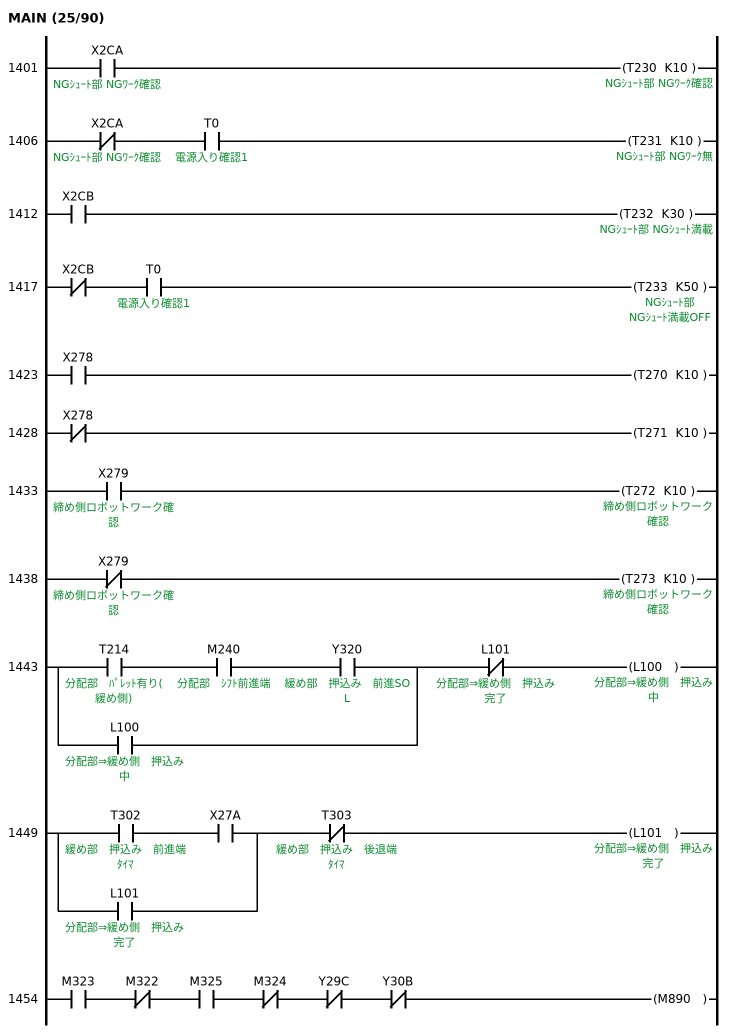
[picture p24: ladder of MAIN, rungs at steps 1401 to 1454]
1401  LD      X2CA  ; NGｼｭｰﾄ部 NGﾜｰｸ確認
      OUT     T230 K10  ; NGｼｭｰﾄ部 NGﾜｰｸ確認
1406  LDI     X2CA  ; NGｼｭｰﾄ部 NGﾜｰｸ確認
      AND     T0  ; 電源入り確認1
      OUT     T231 K10  ; NGｼｭｰﾄ部 NGﾜｰｸ無
1412  LD      X2CB
      OUT     T232 K30  ; NGｼｭｰﾄ部 NGｼｭｰﾄ満載
1417  LDI     X2CB
      AND     T0  ; 電源入り確認1
      OUT     T233 K50  ; NGｼｭｰﾄ部 NGｼｭｰﾄ満載OFF
1423  LD      X278
      OUT     T270 K10
1428  LDI     X278
      OUT     T271 K10
1433  LD      X279  ; 締め側ロボットワーク確認
      OUT     T272 K10  ; 締め側ロボットワーク確認
1438  LDI     X279  ; 締め側ロボットワーク確認
      OUT     T273 K10  ; 締め側ロボットワーク確認
1443  LD      T214  ; 分配部　ﾊﾟﾚｯﾄ有り(緩め側)
      AND     M240  ; 分配部　ｼﾌﾄ前進端
      AND     Y320  ; 緩め部　押込み　前進SOL
      OR      L100  ; 分配部⇒緩め側　押込み中
      ANI     L101  ; 分配部⇒緩め側　押込み完了
      OUT     L100  ; 分配部⇒緩め側　押込み中
1449  LD      T302  ; 緩め部　押込み　前進端　ﾀｲﾏ
      AND     X27A
      OR      L101  ; 分配部⇒緩め側　押込み完了
      ANI     T303  ; 緩め部　押込み　後退端　ﾀｲﾏ
      OUT     L101  ; 分配部⇒緩め側　押込み完了
1454  LD      M323
      ANI     M322
      AND     M325
      ANI     M324
      ANI     Y29C
      ANI     Y30B
      OUT     M890
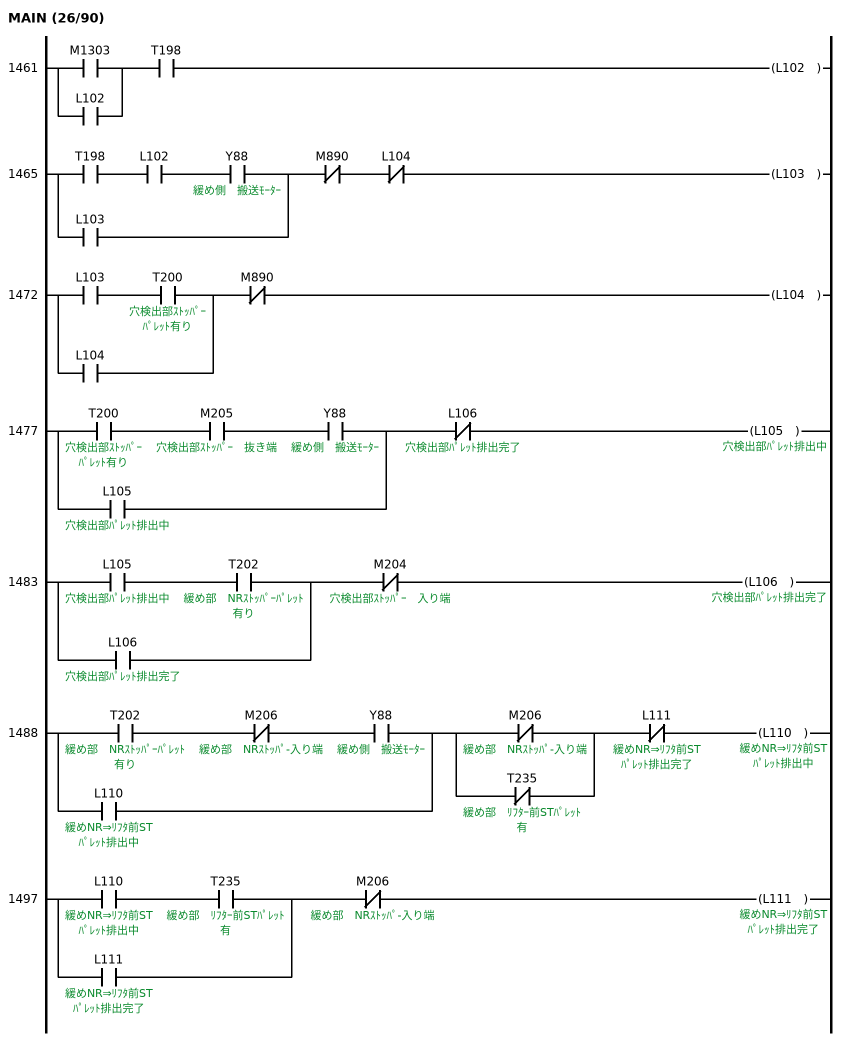
1461  LD      M1303
      OR      L102
      AND     T198
      OUT     L102
1465  LD      T198
      AND     L102
      AND     Y88  ; 緩め側　搬送ﾓｰﾀｰ
      OR      L103
      ANI     M890
      ANI     L104
      OUT     L103
1472  LD      L103
      AND     T200  ; 穴検出部ｽﾄｯﾊﾟｰ 　ﾊﾟﾚｯﾄ有り
      OR      L104
      ANI     M890
      OUT     L104
1477  LD      T200  ; 穴検出部ｽﾄｯﾊﾟｰ 　ﾊﾟﾚｯﾄ有り
      AND     M205  ; 穴検出部ｽﾄｯﾊﾟｰ　抜き端
      AND     Y88  ; 緩め側　搬送ﾓｰﾀｰ
      OR      L105  ; 穴検出部ﾊﾟﾚｯﾄ排出中
      ANI     L106  ; 穴検出部ﾊﾟﾚｯﾄ排出完了
      OUT     L105  ; 穴検出部ﾊﾟﾚｯﾄ排出中
1483  LD      L105  ; 穴検出部ﾊﾟﾚｯﾄ排出中
      AND     T202  ; 緩め部　NRｽﾄｯﾊﾟｰﾊﾟﾚｯﾄ有り
      OR      L106  ; 穴検出部ﾊﾟﾚｯﾄ排出完了
      ANI     M204  ; 穴検出部ｽﾄｯﾊﾟｰ　入り端
      OUT     L106  ; 穴検出部ﾊﾟﾚｯﾄ排出完了
1488  LD      T202  ; 緩め部　NRｽﾄｯﾊﾟｰﾊﾟﾚｯﾄ有り
      ANI     M206  ; 緩め部　NRｽﾄｯﾊﾟ-入り端
      AND     Y88  ; 緩め側　搬送ﾓｰﾀｰ
      OR      L110  ; 緩めNR⇒ﾘﾌﾀ前ST ﾊﾟﾚｯﾄ排出中
      LDI     M206  ; 緩め部　NRｽﾄｯﾊﾟ-入り端
      ORI     T235  ; 緩め部　ﾘﾌﾀｰ前STﾊﾟﾚｯﾄ有
      ANB
      ANI     L111  ; 緩めNR⇒ﾘﾌﾀ前ST ﾊﾟﾚｯﾄ排出完了
      OUT     L110  ; 緩めNR⇒ﾘﾌﾀ前ST ﾊﾟﾚｯﾄ排出中
1497  LD      L110  ; 緩めNR⇒ﾘﾌﾀ前ST ﾊﾟﾚｯﾄ排出中
      AND     T235  ; 緩め部　ﾘﾌﾀｰ前STﾊﾟﾚｯﾄ有
      OR      L111  ; 緩めNR⇒ﾘﾌﾀ前ST ﾊﾟﾚｯﾄ排出完了
      ANI     M206  ; 緩め部　NRｽﾄｯﾊﾟ-入り端
      OUT     L111  ; 緩めNR⇒ﾘﾌﾀ前ST ﾊﾟﾚｯﾄ排出完了
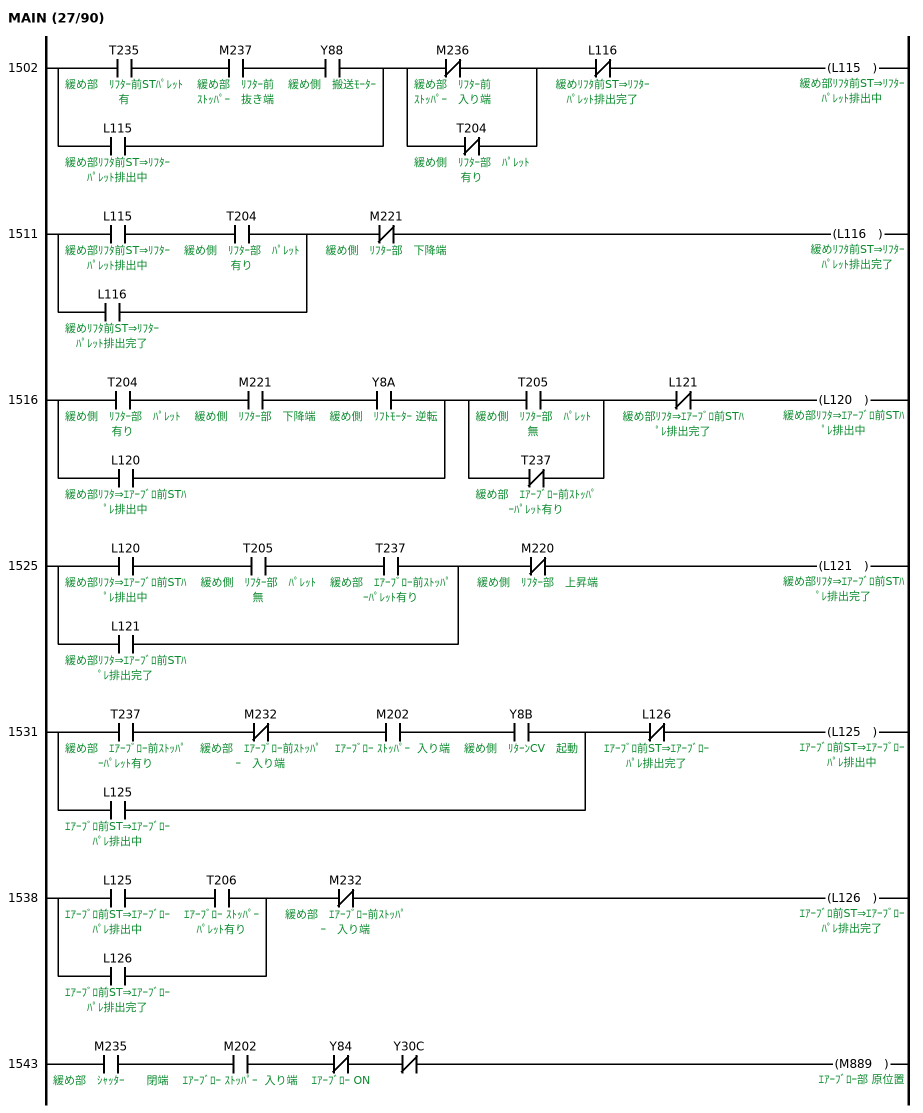
1502  LD      T235  ; 緩め部　ﾘﾌﾀｰ前STﾊﾟﾚｯﾄ有
      AND     M237  ; 緩め部　ﾘﾌﾀｰ前  ｽﾄｯﾊﾟｰ　抜き端
      AND     Y88  ; 緩め側　搬送ﾓｰﾀｰ
      OR      L115  ; 緩め部ﾘﾌﾀ前ST⇒ﾘﾌﾀｰ ﾊﾟﾚｯﾄ排出中
      LDI     M236  ; 緩め部　ﾘﾌﾀｰ前  ｽﾄｯﾊﾟｰ　入り端
      ORI     T204  ; 緩め側　ﾘﾌﾀｰ部　ﾊﾟﾚｯﾄ有り
      ANB
      ANI     L116  ; 緩めﾘﾌﾀ前ST⇒ﾘﾌﾀｰ ﾊﾟﾚｯﾄ排出完了
      OUT     L115  ; 緩め部ﾘﾌﾀ前ST⇒ﾘﾌﾀｰ ﾊﾟﾚｯﾄ排出中
1511  LD      L115  ; 緩め部ﾘﾌﾀ前ST⇒ﾘﾌﾀｰ ﾊﾟﾚｯﾄ排出中
      AND     T204  ; 緩め側　ﾘﾌﾀｰ部　ﾊﾟﾚｯﾄ有り
      OR      L116  ; 緩めﾘﾌﾀ前ST⇒ﾘﾌﾀｰ ﾊﾟﾚｯﾄ排出完了
      ANI     M221  ; 緩め側　ﾘﾌﾀｰ部　下降端
      OUT     L116  ; 緩めﾘﾌﾀ前ST⇒ﾘﾌﾀｰ ﾊﾟﾚｯﾄ排出完了
1516  LD      T204  ; 緩め側　ﾘﾌﾀｰ部　ﾊﾟﾚｯﾄ有り
      AND     M221  ; 緩め側　ﾘﾌﾀｰ部　下降端
      AND     Y8A  ; 緩め側　ﾘﾌﾄﾓｰﾀｰ 逆転
      OR      L120  ; 緩め部ﾘﾌﾀ⇒ｴｱｰﾌﾞﾛ前STﾊﾟﾚ排出中
      LD      T205  ; 緩め側　ﾘﾌﾀｰ部　ﾊﾟﾚｯﾄ無
      ORI     T237  ; 緩め部　ｴｱｰﾌﾞﾛｰ前ｽﾄｯﾊﾟｰﾊﾟﾚｯﾄ有り
      ANB
      ANI     L121  ; 緩め部ﾘﾌﾀ⇒ｴｱｰﾌﾞﾛ前STﾊﾟﾚ排出完了
      OUT     L120  ; 緩め部ﾘﾌﾀ⇒ｴｱｰﾌﾞﾛ前STﾊﾟﾚ排出中
1525  LD      L120  ; 緩め部ﾘﾌﾀ⇒ｴｱｰﾌﾞﾛ前STﾊﾟﾚ排出中
      AND     T205  ; 緩め側　ﾘﾌﾀｰ部　ﾊﾟﾚｯﾄ無
      AND     T237  ; 緩め部　ｴｱｰﾌﾞﾛｰ前ｽﾄｯﾊﾟｰﾊﾟﾚｯﾄ有り
      OR      L121  ; 緩め部ﾘﾌﾀ⇒ｴｱｰﾌﾞﾛ前STﾊﾟﾚ排出完了
      ANI     M220  ; 緩め側　ﾘﾌﾀｰ部　上昇端
      OUT     L121  ; 緩め部ﾘﾌﾀ⇒ｴｱｰﾌﾞﾛ前STﾊﾟﾚ排出完了
1531  LD      T237  ; 緩め部　ｴｱｰﾌﾞﾛｰ前ｽﾄｯﾊﾟｰﾊﾟﾚｯﾄ有り
      ANI     M232  ; 緩め部　ｴｱｰﾌﾞﾛｰ前ｽﾄｯﾊﾟｰ　入り端
      AND     M202  ; ｴｱｰﾌﾞﾛｰ ｽﾄｯﾊﾟｰ  入り端
      AND     Y8B  ; 緩め側　ﾘﾀｰﾝCV　起動
      OR      L125  ; ｴｱｰﾌﾞﾛ前ST⇒ｴｱｰﾌﾞﾛｰ ﾊﾟﾚ排出中
      ANI     L126  ; ｴｱｰﾌﾞﾛ前ST⇒ｴｱｰﾌﾞﾛｰ ﾊﾟﾚ排出完了
      OUT     L125  ; ｴｱｰﾌﾞﾛ前ST⇒ｴｱｰﾌﾞﾛｰ ﾊﾟﾚ排出中
1538  LD      L125  ; ｴｱｰﾌﾞﾛ前ST⇒ｴｱｰﾌﾞﾛｰ ﾊﾟﾚ排出中
      AND     T206  ; ｴｱｰﾌﾞﾛｰ ｽﾄｯﾊﾟｰ  ﾊﾟﾚｯﾄ有り
      OR      L126  ; ｴｱｰﾌﾞﾛ前ST⇒ｴｱｰﾌﾞﾛｰ ﾊﾟﾚ排出完了
      ANI     M232  ; 緩め部　ｴｱｰﾌﾞﾛｰ前ｽﾄｯﾊﾟｰ　入り端
      OUT     L126  ; ｴｱｰﾌﾞﾛ前ST⇒ｴｱｰﾌﾞﾛｰ ﾊﾟﾚ排出完了
1543  LD      M235  ; 緩め部　ｼｬｯﾀｰ　　閉端
      AND     M202  ; ｴｱｰﾌﾞﾛｰ ｽﾄｯﾊﾟｰ  入り端
      ANI     Y84  ; ｴｱｰﾌﾞﾛｰ ON
      ANI     Y30C
      OUT     M889  ; ｴｱｰﾌﾞﾛｰ部 原位置
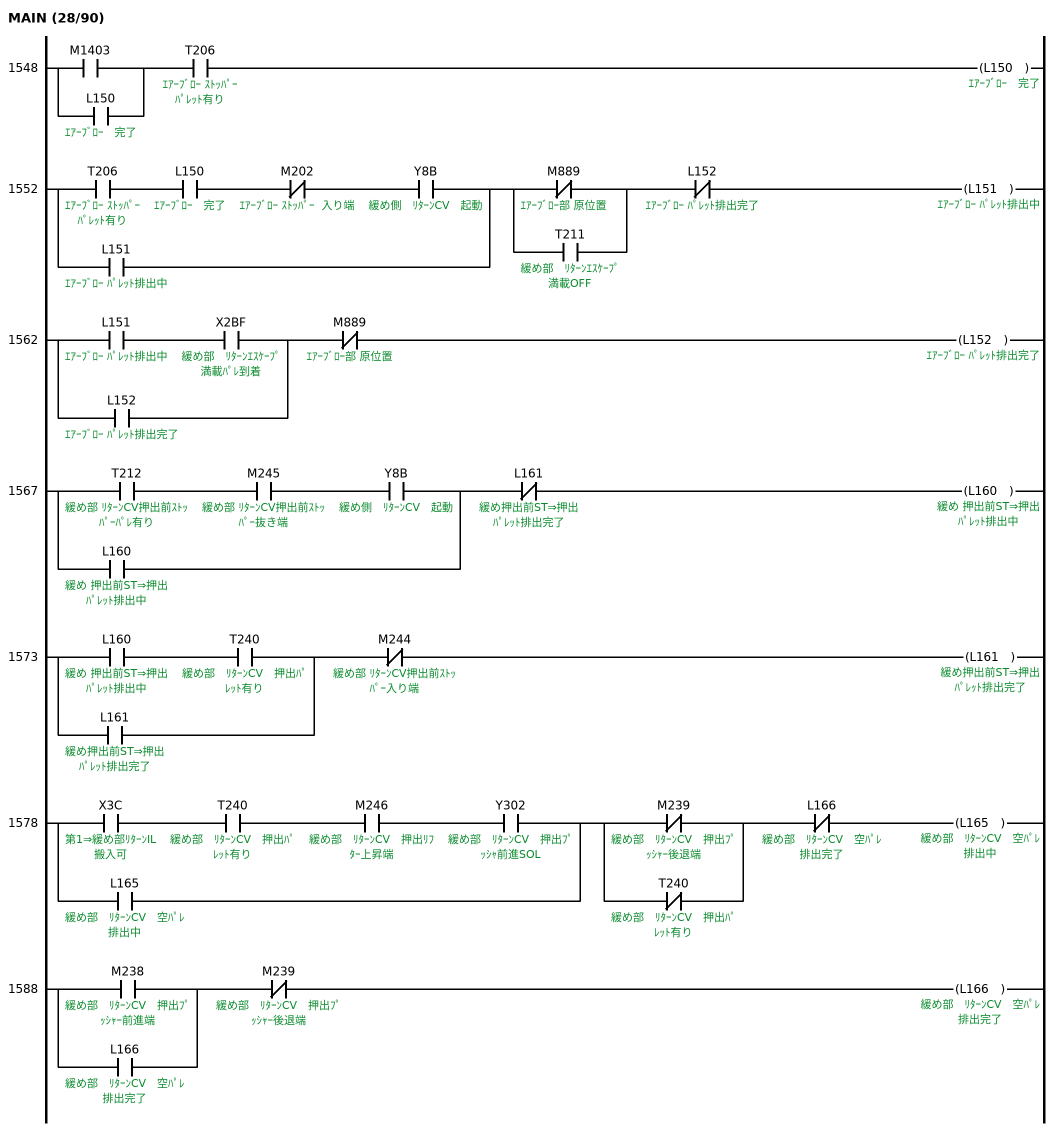
1548  LD      M1403
      OR      L150  ; ｴｱｰﾌﾞﾛｰ　完了
      AND     T206  ; ｴｱｰﾌﾞﾛｰ ｽﾄｯﾊﾟｰ  ﾊﾟﾚｯﾄ有り
      OUT     L150  ; ｴｱｰﾌﾞﾛｰ　完了
1552  LD      T206  ; ｴｱｰﾌﾞﾛｰ ｽﾄｯﾊﾟｰ  ﾊﾟﾚｯﾄ有り
      AND     L150  ; ｴｱｰﾌﾞﾛｰ　完了
      ANI     M202  ; ｴｱｰﾌﾞﾛｰ ｽﾄｯﾊﾟｰ  入り端
      AND     Y8B  ; 緩め側　ﾘﾀｰﾝCV　起動
      OR      L151  ; ｴｱｰﾌﾞﾛｰ ﾊﾟﾚｯﾄ排出中
      LDI     M889  ; ｴｱｰﾌﾞﾛｰ部 原位置
      OR      T211  ; 緩め部　ﾘﾀｰﾝｴｽｹｰﾌﾟ 満載OFF
      ANB
      ANI     L152  ; ｴｱｰﾌﾞﾛｰ ﾊﾟﾚｯﾄ排出完了
      OUT     L151  ; ｴｱｰﾌﾞﾛｰ ﾊﾟﾚｯﾄ排出中
1562  LD      L151  ; ｴｱｰﾌﾞﾛｰ ﾊﾟﾚｯﾄ排出中
      AND     X2BF  ; 緩め部　ﾘﾀｰﾝｴｽｹｰﾌﾟ 満載ﾊﾟﾚ到着
      OR      L152  ; ｴｱｰﾌﾞﾛｰ ﾊﾟﾚｯﾄ排出完了
      ANI     M889  ; ｴｱｰﾌﾞﾛｰ部 原位置
      OUT     L152  ; ｴｱｰﾌﾞﾛｰ ﾊﾟﾚｯﾄ排出完了
1567  LD      T212  ; 緩め部 ﾘﾀｰﾝCV押出前ｽﾄｯﾊﾟｰﾊﾟﾚ有り
      AND     M245  ; 緩め部 ﾘﾀｰﾝCV押出前ｽﾄｯﾊﾟｰ抜き端
      AND     Y8B  ; 緩め側　ﾘﾀｰﾝCV　起動
      OR      L160  ; 緩め 押出前ST⇒押出 ﾊﾟﾚｯﾄ排出中
      ANI     L161  ; 緩め押出前ST⇒押出 ﾊﾟﾚｯﾄ排出完了
      OUT     L160  ; 緩め 押出前ST⇒押出 ﾊﾟﾚｯﾄ排出中
1573  LD      L160  ; 緩め 押出前ST⇒押出 ﾊﾟﾚｯﾄ排出中
      AND     T240  ; 緩め部　ﾘﾀｰﾝCV　押出ﾊﾟﾚｯﾄ有り
      OR      L161  ; 緩め押出前ST⇒押出 ﾊﾟﾚｯﾄ排出完了
      ANI     M244  ; 緩め部 ﾘﾀｰﾝCV押出前ｽﾄｯﾊﾟｰ入り端
      OUT     L161  ; 緩め押出前ST⇒押出 ﾊﾟﾚｯﾄ排出完了
1578  LD      X3C  ; 第1⇒緩め部ﾘﾀｰﾝIL 搬入可
      AND     T240  ; 緩め部　ﾘﾀｰﾝCV　押出ﾊﾟﾚｯﾄ有り
      AND     M246  ; 緩め部　ﾘﾀｰﾝCV　押出ﾘﾌﾀｰ上昇端
      AND     Y302  ; 緩め部　ﾘﾀｰﾝCV　押出ﾌﾟｯｼｬ前進SOL
      OR      L165  ; 緩め部　ﾘﾀｰﾝCV　空ﾊﾟﾚ排出中
      LDI     M239  ; 緩め部　ﾘﾀｰﾝCV　押出ﾌﾟｯｼｬｰ後退端
      ORI     T240  ; 緩め部　ﾘﾀｰﾝCV　押出ﾊﾟﾚｯﾄ有り
      ANB
      ANI     L166  ; 緩め部　ﾘﾀｰﾝCV　空ﾊﾟﾚ排出完了
      OUT     L165  ; 緩め部　ﾘﾀｰﾝCV　空ﾊﾟﾚ排出中
1588  LD      M238  ; 緩め部　ﾘﾀｰﾝCV　押出ﾌﾟｯｼｬｰ前進端
      OR      L166  ; 緩め部　ﾘﾀｰﾝCV　空ﾊﾟﾚ排出完了
      ANI     M239  ; 緩め部　ﾘﾀｰﾝCV　押出ﾌﾟｯｼｬｰ後退端
      OUT     L166  ; 緩め部　ﾘﾀｰﾝCV　空ﾊﾟﾚ排出完了
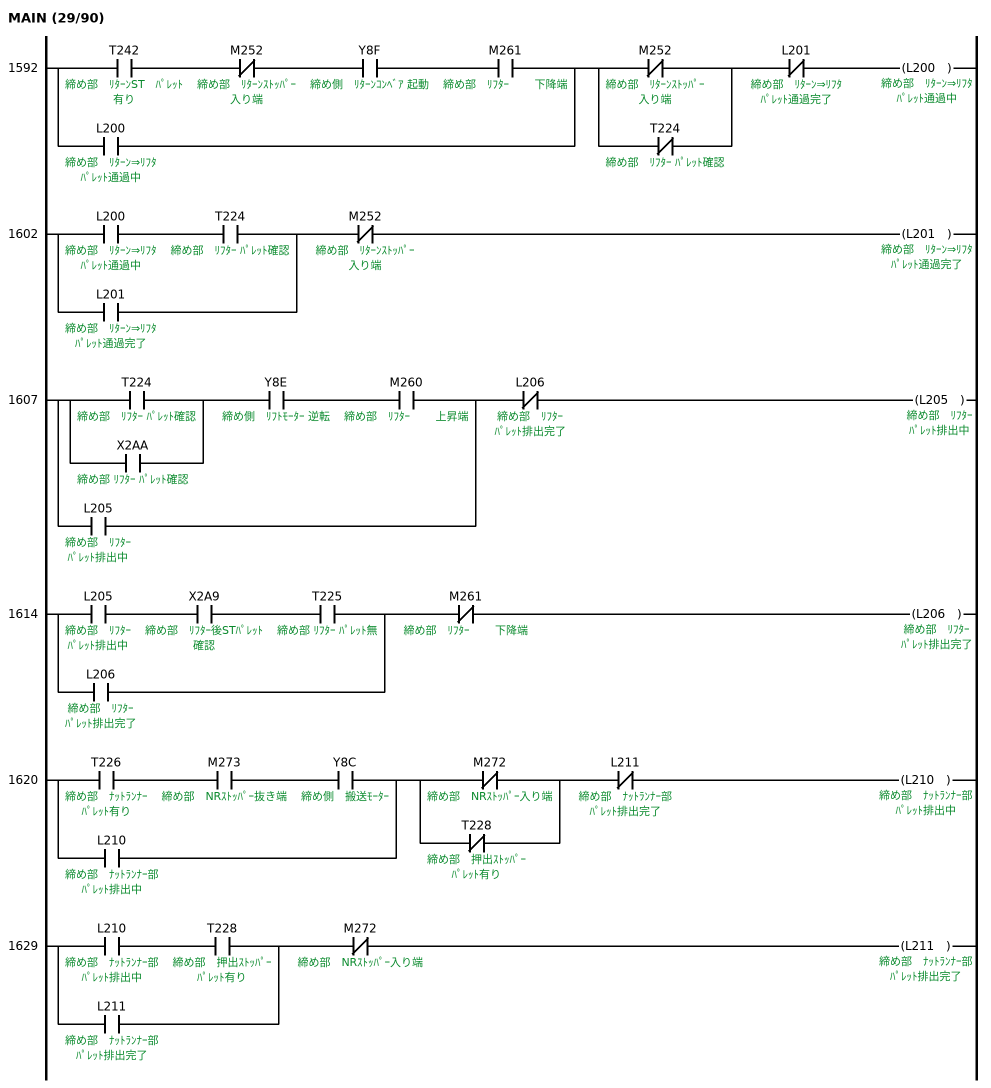
1592  LD      T242  ; 締め部　ﾘﾀｰﾝST　ﾊﾟﾚｯﾄ有り
      ANI     M252  ; 締め部　ﾘﾀｰﾝｽﾄｯﾊﾟｰ 入り端
      AND     Y8F  ; 締め側　ﾘﾀｰﾝｺﾝﾍﾞｱ 起動
      AND     M261  ; 締め部　ﾘﾌﾀｰ 　　下降端
      OR      L200  ; 締め部　ﾘﾀｰﾝ⇒ﾘﾌﾀ ﾊﾟﾚｯﾄ通過中
      LDI     M252  ; 締め部　ﾘﾀｰﾝｽﾄｯﾊﾟｰ 入り端
      ORI     T224  ; 締め部　ﾘﾌﾀｰ ﾊﾟﾚｯﾄ確認
      ANB
      ANI     L201  ; 締め部　ﾘﾀｰﾝ⇒ﾘﾌﾀ ﾊﾟﾚｯﾄ通過完了
      OUT     L200  ; 締め部　ﾘﾀｰﾝ⇒ﾘﾌﾀ ﾊﾟﾚｯﾄ通過中
1602  LD      L200  ; 締め部　ﾘﾀｰﾝ⇒ﾘﾌﾀ ﾊﾟﾚｯﾄ通過中
      AND     T224  ; 締め部　ﾘﾌﾀｰ ﾊﾟﾚｯﾄ確認
      OR      L201  ; 締め部　ﾘﾀｰﾝ⇒ﾘﾌﾀ ﾊﾟﾚｯﾄ通過完了
      ANI     M252  ; 締め部　ﾘﾀｰﾝｽﾄｯﾊﾟｰ 入り端
      OUT     L201  ; 締め部　ﾘﾀｰﾝ⇒ﾘﾌﾀ ﾊﾟﾚｯﾄ通過完了
1607  LD      T224  ; 締め部　ﾘﾌﾀｰ ﾊﾟﾚｯﾄ確認
      OR      X2AA  ; 締め部 ﾘﾌﾀｰ ﾊﾟﾚｯﾄ確認
      AND     Y8E  ; 締め側　ﾘﾌﾄﾓｰﾀｰ 逆転
      AND     M260  ; 締め部　ﾘﾌﾀｰ 　　上昇端
      OR      L205  ; 締め部　ﾘﾌﾀｰ ﾊﾟﾚｯﾄ排出中
      ANI     L206  ; 締め部　ﾘﾌﾀｰ ﾊﾟﾚｯﾄ排出完了
      OUT     L205  ; 締め部　ﾘﾌﾀｰ ﾊﾟﾚｯﾄ排出中
1614  LD      L205  ; 締め部　ﾘﾌﾀｰ ﾊﾟﾚｯﾄ排出中
      AND     X2A9  ; 締め部　ﾘﾌﾀｰ後STﾊﾟﾚｯﾄ確認
      AND     T225  ; 締め部 ﾘﾌﾀｰ ﾊﾟﾚｯﾄ無
      OR      L206  ; 締め部　ﾘﾌﾀｰ ﾊﾟﾚｯﾄ排出完了
      ANI     M261  ; 締め部　ﾘﾌﾀｰ 　　下降端
      OUT     L206  ; 締め部　ﾘﾌﾀｰ ﾊﾟﾚｯﾄ排出完了
1620  LD      T226  ; 締め部　ﾅｯﾄﾗﾝﾅｰ ﾊﾟﾚｯﾄ有り
      AND     M273  ; 締め部　NRｽﾄｯﾊﾟｰ抜き端
      AND     Y8C  ; 締め側　搬送ﾓｰﾀｰ
      OR      L210  ; 締め部　ﾅｯﾄﾗﾝﾅｰ部 ﾊﾟﾚｯﾄ排出中
      LDI     M272  ; 締め部　NRｽﾄｯﾊﾟｰ入り端
      ORI     T228  ; 締め部　押出ｽﾄｯﾊﾟｰ ﾊﾟﾚｯﾄ有り
      ANB
      ANI     L211  ; 締め部　ﾅｯﾄﾗﾝﾅｰ部 ﾊﾟﾚｯﾄ排出完了
      OUT     L210  ; 締め部　ﾅｯﾄﾗﾝﾅｰ部 ﾊﾟﾚｯﾄ排出中
1629  LD      L210  ; 締め部　ﾅｯﾄﾗﾝﾅｰ部 ﾊﾟﾚｯﾄ排出中
      AND     T228  ; 締め部　押出ｽﾄｯﾊﾟｰ ﾊﾟﾚｯﾄ有り
      OR      L211  ; 締め部　ﾅｯﾄﾗﾝﾅｰ部 ﾊﾟﾚｯﾄ排出完了
      ANI     M272  ; 締め部　NRｽﾄｯﾊﾟｰ入り端
      OUT     L211  ; 締め部　ﾅｯﾄﾗﾝﾅｰ部 ﾊﾟﾚｯﾄ排出完了
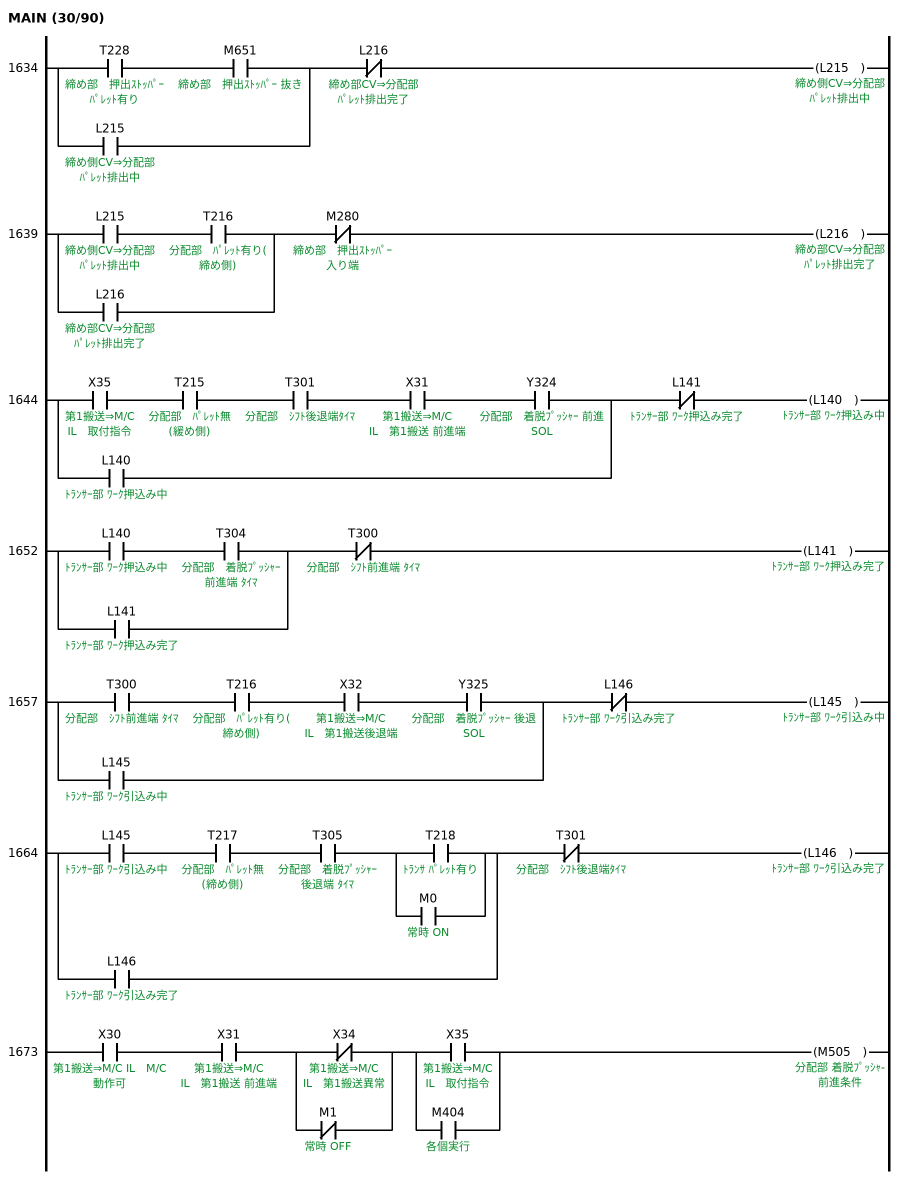
1634  LD      T228  ; 締め部　押出ｽﾄｯﾊﾟｰ ﾊﾟﾚｯﾄ有り
      AND     M651  ; 締め部　押出ｽﾄｯﾊﾟｰ 抜き
      OR      L215  ; 締め側CV⇒分配部 ﾊﾟﾚｯﾄ排出中
      ANI     L216  ; 締め部CV⇒分配部 ﾊﾟﾚｯﾄ排出完了
      OUT     L215  ; 締め側CV⇒分配部 ﾊﾟﾚｯﾄ排出中
1639  LD      L215  ; 締め側CV⇒分配部 ﾊﾟﾚｯﾄ排出中
      AND     T216  ; 分配部　ﾊﾟﾚｯﾄ有り(締め側)
      OR      L216  ; 締め部CV⇒分配部 ﾊﾟﾚｯﾄ排出完了
      ANI     M280  ; 締め部　押出ｽﾄｯﾊﾟｰ 入り端
      OUT     L216  ; 締め部CV⇒分配部 ﾊﾟﾚｯﾄ排出完了
1644  LD      X35  ; 第1搬送⇒M/C IL　取付指令
      AND     T215  ; 分配部　ﾊﾟﾚｯﾄ無 (緩め側)
      AND     T301  ; 分配部　ｼﾌﾄ後退端ﾀｲﾏ
      AND     X31  ; 第1搬送⇒M/C IL　第1搬送 前進端
      AND     Y324  ; 分配部　着脱ﾌﾟｯｼｬｰ 前進 SOL
      OR      L140  ; ﾄﾗﾝｻｰ部 ﾜｰｸ押込み中
      ANI     L141  ; ﾄﾗﾝｻｰ部 ﾜｰｸ押込み完了
      OUT     L140  ; ﾄﾗﾝｻｰ部 ﾜｰｸ押込み中
1652  LD      L140  ; ﾄﾗﾝｻｰ部 ﾜｰｸ押込み中
      AND     T304  ; 分配部　着脱ﾌﾟｯｼｬｰ 前進端 ﾀｲﾏ
      OR      L141  ; ﾄﾗﾝｻｰ部 ﾜｰｸ押込み完了
      ANI     T300  ; 分配部　ｼﾌﾄ前進端 ﾀｲﾏ
      OUT     L141  ; ﾄﾗﾝｻｰ部 ﾜｰｸ押込み完了
1657  LD      T300  ; 分配部　ｼﾌﾄ前進端 ﾀｲﾏ
      AND     T216  ; 分配部　ﾊﾟﾚｯﾄ有り(締め側)
      AND     X32  ; 第1搬送⇒M/C IL　第1搬送後退端
      AND     Y325  ; 分配部　着脱ﾌﾟｯｼｬｰ 後退 SOL
      OR      L145  ; ﾄﾗﾝｻｰ部 ﾜｰｸ引込み中
      ANI     L146  ; ﾄﾗﾝｻｰ部 ﾜｰｸ引込み完了
      OUT     L145  ; ﾄﾗﾝｻｰ部 ﾜｰｸ引込み中
1664  LD      L145  ; ﾄﾗﾝｻｰ部 ﾜｰｸ引込み中
      AND     T217  ; 分配部　ﾊﾟﾚｯﾄ無 (締め側)
      AND     T305  ; 分配部　着脱ﾌﾟｯｼｬｰ 後退端 ﾀｲﾏ
      LD      T218  ; ﾄﾗﾝｻ ﾊﾟﾚｯﾄ有り
      OR      M0  ; 常時 ON
      ANB
      OR      L146  ; ﾄﾗﾝｻｰ部 ﾜｰｸ引込み完了
      ANI     T301  ; 分配部　ｼﾌﾄ後退端ﾀｲﾏ
      OUT     L146  ; ﾄﾗﾝｻｰ部 ﾜｰｸ引込み完了
1673  LD      X30  ; 第1搬送⇒M/C IL　M/C 動作可
      AND     X31  ; 第1搬送⇒M/C IL　第1搬送 前進端
      LDI     X34  ; 第1搬送⇒M/C IL　第1搬送異常
      ORI     M1  ; 常時 OFF
      ANB
      LD      X35  ; 第1搬送⇒M/C IL　取付指令
      OR      M404  ; 各個実行
      ANB
      OUT     M505  ; 分配部 着脱ﾌﾟｯｼｬ- 前進条件
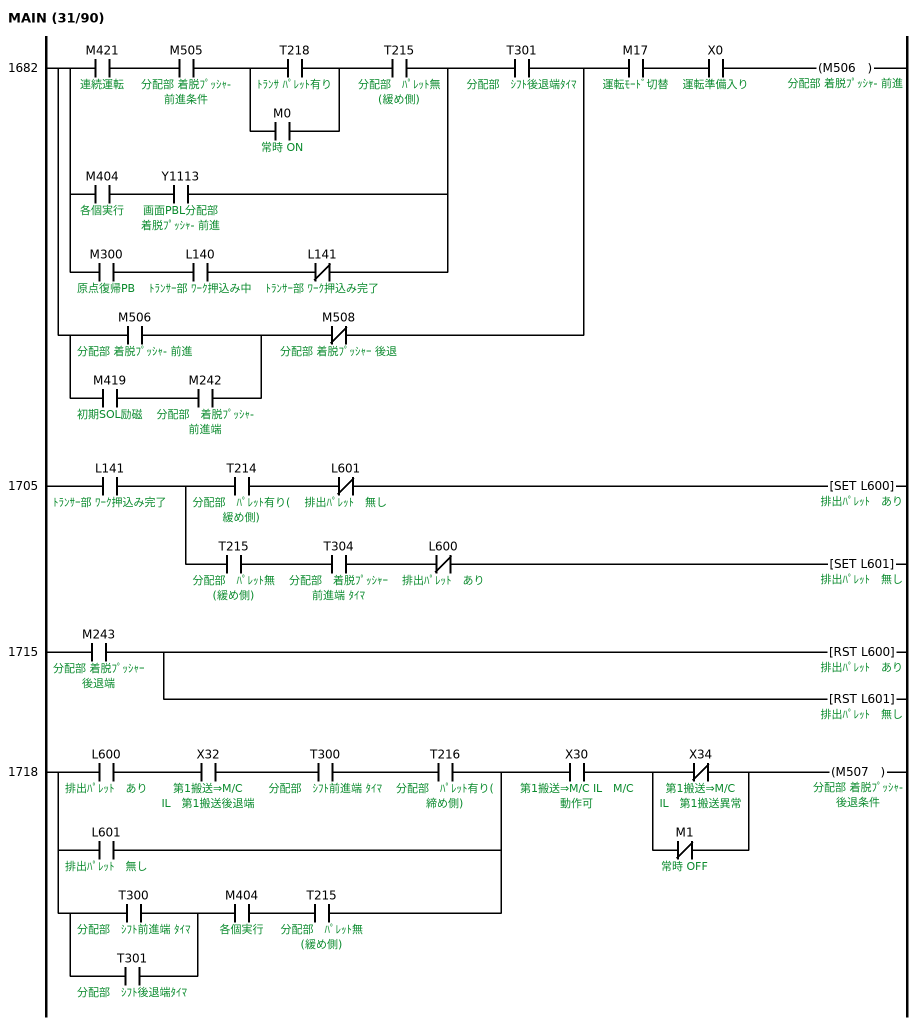
1682  LD      M421  ; 連続運転
      AND     M505  ; 分配部 着脱ﾌﾟｯｼｬ- 前進条件
      LD      T218  ; ﾄﾗﾝｻ ﾊﾟﾚｯﾄ有り
      OR      M0  ; 常時 ON
      ANB
      AND     T215  ; 分配部　ﾊﾟﾚｯﾄ無 (緩め側)
      LD      M404  ; 各個実行
      AND     Y1113  ; 画面PBL分配部 着脱ﾌﾟｯｼｬ- 前進
      ORB
      LD      M300  ; 原点復帰PB
      AND     L140  ; ﾄﾗﾝｻｰ部 ﾜｰｸ押込み中
      ANI     L141  ; ﾄﾗﾝｻｰ部 ﾜｰｸ押込み完了
      ORB
      AND     T301  ; 分配部　ｼﾌﾄ後退端ﾀｲﾏ
      LD      M506  ; 分配部 着脱ﾌﾟｯｼｬ- 前進
      LD      M419  ; 初期SOL励磁
      AND     M242  ; 分配部　着脱ﾌﾟｯｼｬ- 前進端
      ORB
      ANI     M508  ; 分配部 着脱ﾌﾟｯｼｬｰ 後退
      ORB
      AND     M17  ; 運転ﾓｰﾄﾞ切替
      AND     X0  ; 運転準備入り
      OUT     M506  ; 分配部 着脱ﾌﾟｯｼｬ- 前進
1705  LD      L141  ; ﾄﾗﾝｻｰ部 ﾜｰｸ押込み完了
      MPS
      AND     T214  ; 分配部　ﾊﾟﾚｯﾄ有り(緩め側)
      ANI     L601  ; 排出ﾊﾟﾚｯﾄ　無し
      SET     L600  ; 排出ﾊﾟﾚｯﾄ　あり
      MPP
      AND     T215  ; 分配部　ﾊﾟﾚｯﾄ無 (緩め側)
      AND     T304  ; 分配部　着脱ﾌﾟｯｼｬｰ 前進端 ﾀｲﾏ
      ANI     L600  ; 排出ﾊﾟﾚｯﾄ　あり
      SET     L601  ; 排出ﾊﾟﾚｯﾄ　無し
1715  LD      M243  ; 分配部 着脱ﾌﾟｯｼｬｰ 後退端
      RST     L600  ; 排出ﾊﾟﾚｯﾄ　あり
      RST     L601  ; 排出ﾊﾟﾚｯﾄ　無し
1718  LD      L600  ; 排出ﾊﾟﾚｯﾄ　あり
      AND     X32  ; 第1搬送⇒M/C IL　第1搬送後退端
      AND     T300  ; 分配部　ｼﾌﾄ前進端 ﾀｲﾏ
      AND     T216  ; 分配部　ﾊﾟﾚｯﾄ有り(締め側)
      OR      L601  ; 排出ﾊﾟﾚｯﾄ　無し
      LD      T300  ; 分配部　ｼﾌﾄ前進端 ﾀｲﾏ
      OR      T301  ; 分配部　ｼﾌﾄ後退端ﾀｲﾏ
      AND     M404  ; 各個実行
      AND     T215  ; 分配部　ﾊﾟﾚｯﾄ無 (緩め側)
      ORB
      AND     X30  ; 第1搬送⇒M/C IL　M/C 動作可
      LDI     X34  ; 第1搬送⇒M/C IL　第1搬送異常
      ORI     M1  ; 常時 OFF
      ANB
      OUT     M507  ; 分配部 着脱ﾌﾟｯｼｬ-後退条件
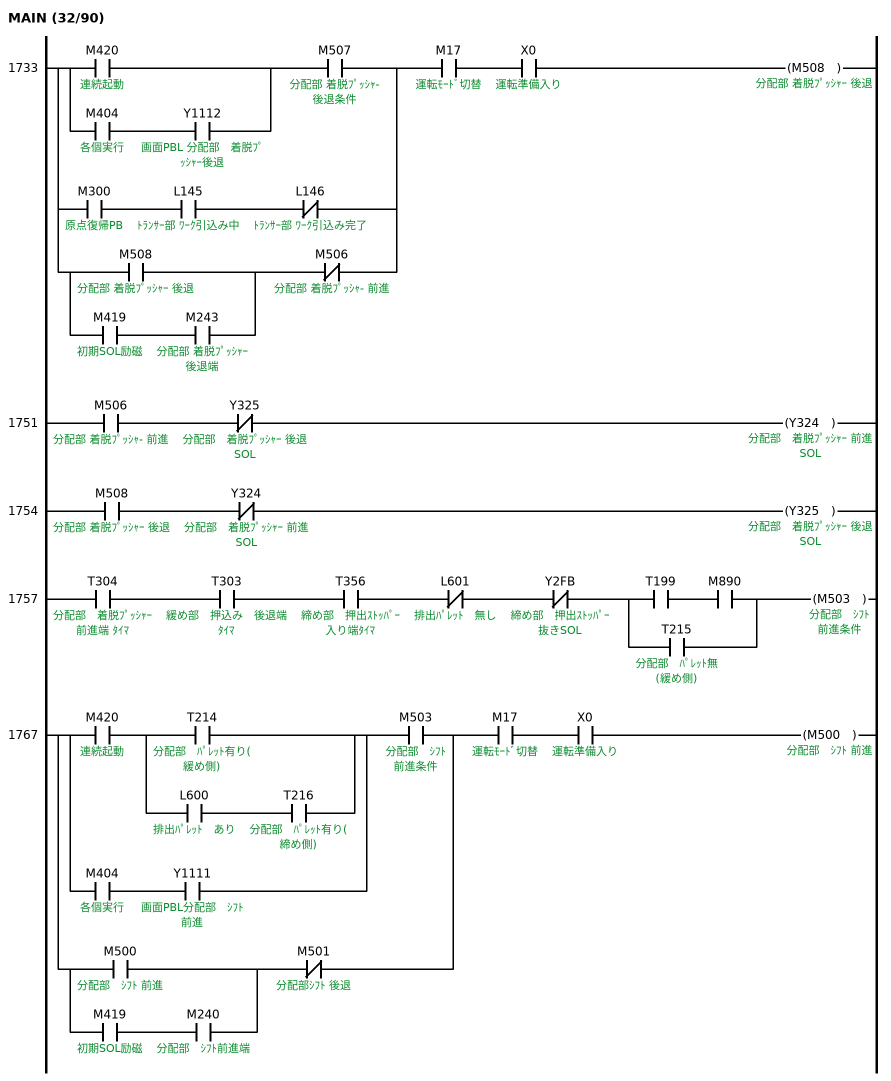
1733  LD      M420  ; 連続起動
      LD      M404  ; 各個実行
      AND     Y1112  ; 画面PBL 分配部　着脱ﾌﾟｯｼｬｰ後退
      ORB
      AND     M507  ; 分配部 着脱ﾌﾟｯｼｬ-後退条件
      LD      M300  ; 原点復帰PB
      AND     L145  ; ﾄﾗﾝｻｰ部 ﾜｰｸ引込み中
      ANI     L146  ; ﾄﾗﾝｻｰ部 ﾜｰｸ引込み完了
      ORB
      LD      M508  ; 分配部 着脱ﾌﾟｯｼｬｰ 後退
      LD      M419  ; 初期SOL励磁
      AND     M243  ; 分配部 着脱ﾌﾟｯｼｬｰ 後退端
      ORB
      ANI     M506  ; 分配部 着脱ﾌﾟｯｼｬ- 前進
      ORB
      AND     M17  ; 運転ﾓｰﾄﾞ切替
      AND     X0  ; 運転準備入り
      OUT     M508  ; 分配部 着脱ﾌﾟｯｼｬｰ 後退
1751  LD      M506  ; 分配部 着脱ﾌﾟｯｼｬ- 前進
      ANI     Y325  ; 分配部　着脱ﾌﾟｯｼｬｰ 後退 SOL
      OUT     Y324  ; 分配部　着脱ﾌﾟｯｼｬｰ 前進 SOL
1754  LD      M508  ; 分配部 着脱ﾌﾟｯｼｬｰ 後退
      ANI     Y324  ; 分配部　着脱ﾌﾟｯｼｬｰ 前進 SOL
      OUT     Y325  ; 分配部　着脱ﾌﾟｯｼｬｰ 後退 SOL
1757  LD      T304  ; 分配部　着脱ﾌﾟｯｼｬｰ 前進端 ﾀｲﾏ
      AND     T303  ; 緩め部　押込み　後退端　ﾀｲﾏ
      AND     T356  ; 締め部　押出ｽﾄｯﾊﾟｰ 入り端ﾀｲﾏ
      ANI     L601  ; 排出ﾊﾟﾚｯﾄ　無し
      ANI     Y2FB  ; 締め部　押出ｽﾄｯﾊﾟｰ 抜きSOL
      LD      T199
      AND     M890
      OR      T215  ; 分配部　ﾊﾟﾚｯﾄ無 (緩め側)
      ANB
      OUT     M503  ; 分配部　ｼﾌﾄ 　　前進条件
1767  LD      M420  ; 連続起動
      LD      T214  ; 分配部　ﾊﾟﾚｯﾄ有り(緩め側)
      LD      L600  ; 排出ﾊﾟﾚｯﾄ　あり
      AND     T216  ; 分配部　ﾊﾟﾚｯﾄ有り(締め側)
      ORB
      ANB
      LD      M404  ; 各個実行
      AND     Y1111  ; 画面PBL分配部　ｼﾌﾄ 前進
      ORB
      AND     M503  ; 分配部　ｼﾌﾄ 　　前進条件
      LD      M500  ; 分配部　ｼﾌﾄ 前進
      LD      M419  ; 初期SOL励磁
      AND     M240  ; 分配部　ｼﾌﾄ前進端
      ORB
      ANI     M501  ; 分配部ｼﾌﾄ 後退
      ORB
      AND     M17  ; 運転ﾓｰﾄﾞ切替
      AND     X0  ; 運転準備入り
      OUT     M500  ; 分配部　ｼﾌﾄ 前進
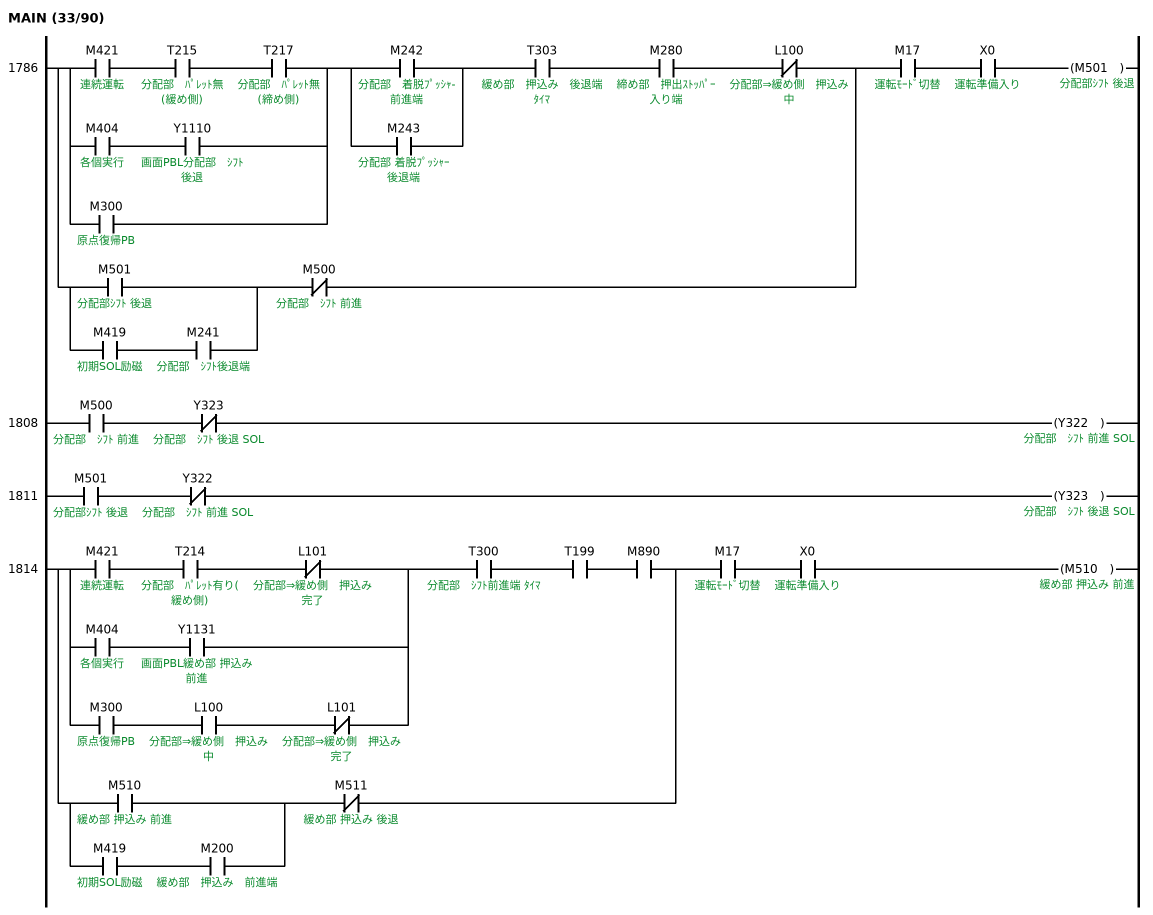
1786  LD      M421  ; 連続運転
      AND     T215  ; 分配部　ﾊﾟﾚｯﾄ無 (緩め側)
      AND     T217  ; 分配部　ﾊﾟﾚｯﾄ無 (締め側)
      LD      M404  ; 各個実行
      AND     Y1110  ; 画面PBL分配部　ｼﾌﾄ 後退
      ORB
      OR      M300  ; 原点復帰PB
      LD      M242  ; 分配部　着脱ﾌﾟｯｼｬ- 前進端
      OR      M243  ; 分配部 着脱ﾌﾟｯｼｬｰ 後退端
      ANB
      AND     T303  ; 緩め部　押込み　後退端　ﾀｲﾏ
      AND     M280  ; 締め部　押出ｽﾄｯﾊﾟｰ 入り端
      ANI     L100  ; 分配部⇒緩め側　押込み中
      LD      M501  ; 分配部ｼﾌﾄ 後退
      LD      M419  ; 初期SOL励磁
      AND     M241  ; 分配部　ｼﾌﾄ後退端
      ORB
      ANI     M500  ; 分配部　ｼﾌﾄ 前進
      ORB
      AND     M17  ; 運転ﾓｰﾄﾞ切替
      AND     X0  ; 運転準備入り
      OUT     M501  ; 分配部ｼﾌﾄ 後退
1808  LD      M500  ; 分配部　ｼﾌﾄ 前進
      ANI     Y323  ; 分配部　ｼﾌﾄ 後退 SOL
      OUT     Y322  ; 分配部　ｼﾌﾄ 前進 SOL
1811  LD      M501  ; 分配部ｼﾌﾄ 後退
      ANI     Y322  ; 分配部　ｼﾌﾄ 前進 SOL
      OUT     Y323  ; 分配部　ｼﾌﾄ 後退 SOL
1814  LD      M421  ; 連続運転
      AND     T214  ; 分配部　ﾊﾟﾚｯﾄ有り(緩め側)
      ANI     L101  ; 分配部⇒緩め側　押込み完了
      LD      M404  ; 各個実行
      AND     Y1131  ; 画面PBL緩め部 押込み 前進
      ORB
      LD      M300  ; 原点復帰PB
      AND     L100  ; 分配部⇒緩め側　押込み中
      ANI     L101  ; 分配部⇒緩め側　押込み完了
      ORB
      AND     T300  ; 分配部　ｼﾌﾄ前進端 ﾀｲﾏ
      AND     T199
      AND     M890
      LD      M510  ; 緩め部 押込み 前進
      LD      M419  ; 初期SOL励磁
      AND     M200  ; 緩め部　押込み　前進端
      ORB
      ANI     M511  ; 緩め部 押込み 後退
      ORB
      AND     M17  ; 運転ﾓｰﾄﾞ切替
      AND     X0  ; 運転準備入り
      OUT     M510  ; 緩め部 押込み 前進
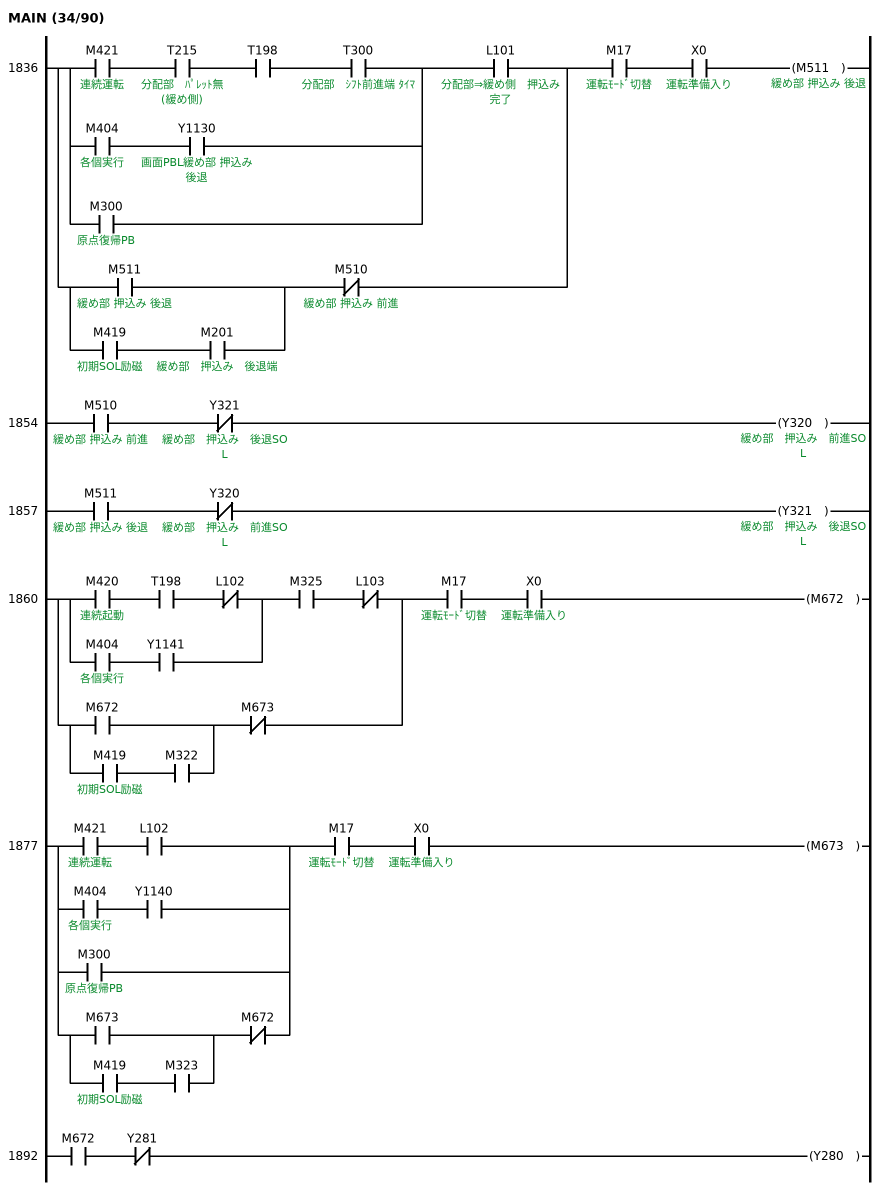
1836  LD      M421  ; 連続運転
      AND     T215  ; 分配部　ﾊﾟﾚｯﾄ無 (緩め側)
      AND     T198
      AND     T300  ; 分配部　ｼﾌﾄ前進端 ﾀｲﾏ
      LD      M404  ; 各個実行
      AND     Y1130  ; 画面PBL緩め部 押込み 後退
      ORB
      OR      M300  ; 原点復帰PB
      AND     L101  ; 分配部⇒緩め側　押込み完了
      LD      M511  ; 緩め部 押込み 後退
      LD      M419  ; 初期SOL励磁
      AND     M201  ; 緩め部　押込み　後退端
      ORB
      ANI     M510  ; 緩め部 押込み 前進
      ORB
      AND     M17  ; 運転ﾓｰﾄﾞ切替
      AND     X0  ; 運転準備入り
      OUT     M511  ; 緩め部 押込み 後退
1854  LD      M510  ; 緩め部 押込み 前進
      ANI     Y321  ; 緩め部　押込み　後退SOL
      OUT     Y320  ; 緩め部　押込み　前進SOL
1857  LD      M511  ; 緩め部 押込み 後退
      ANI     Y320  ; 緩め部　押込み　前進SOL
      OUT     Y321  ; 緩め部　押込み　後退SOL
1860  LD      M420  ; 連続起動
      AND     T198
      ANI     L102
      LD      M404  ; 各個実行
      AND     Y1141
      ORB
      AND     M325
      ANI     L103
      LD      M672
      LD      M419  ; 初期SOL励磁
      AND     M322
      ORB
      ANI     M673
      ORB
      AND     M17  ; 運転ﾓｰﾄﾞ切替
      AND     X0  ; 運転準備入り
      OUT     M672
1877  LD      M421  ; 連続運転
      AND     L102
      LD      M404  ; 各個実行
      AND     Y1140
      ORB
      OR      M300  ; 原点復帰PB
      LD      M673
      LD      M419  ; 初期SOL励磁
      AND     M323
      ORB
      ANI     M672
      ORB
      AND     M17  ; 運転ﾓｰﾄﾞ切替
      AND     X0  ; 運転準備入り
      OUT     M673
1892  LD      M672
      ANI     Y281
      OUT     Y280
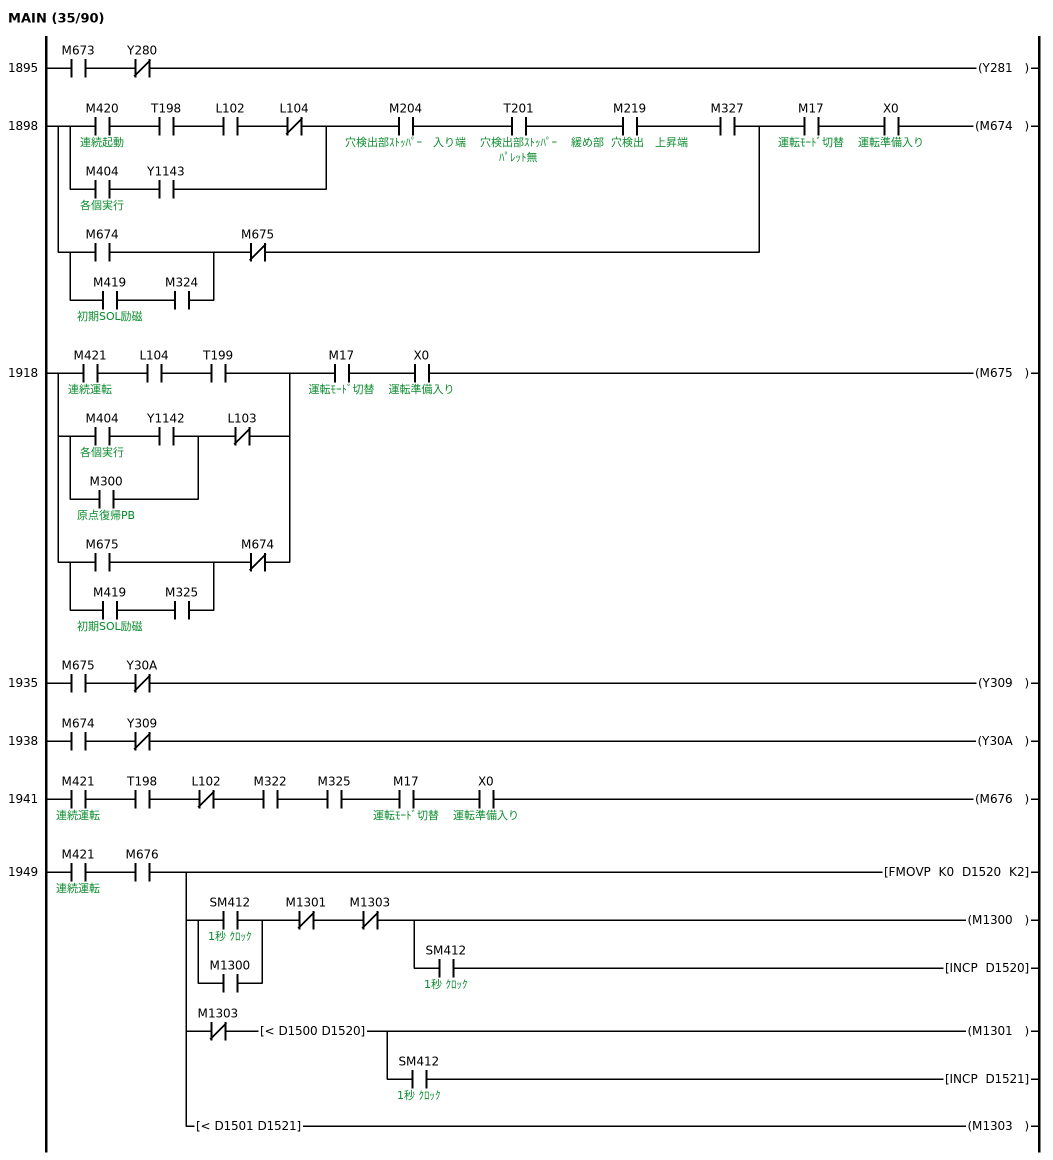
1895  LD      M673
      ANI     Y280
      OUT     Y281
1898  LD      M420  ; 連続起動
      AND     T198
      AND     L102
      ANI     L104
      LD      M404  ; 各個実行
      AND     Y1143
      ORB
      AND     M204  ; 穴検出部ｽﾄｯﾊﾟｰ　入り端
      AND     T201  ; 穴検出部ｽﾄｯﾊﾟｰ 　ﾊﾟﾚｯﾄ無
      AND     M219  ; 緩め部  穴検出　上昇端
      AND     M327
      LD      M674
      LD      M419  ; 初期SOL励磁
      AND     M324
      ORB
      ANI     M675
      ORB
      AND     M17  ; 運転ﾓｰﾄﾞ切替
      AND     X0  ; 運転準備入り
      OUT     M674
1918  LD      M421  ; 連続運転
      AND     L104
      AND     T199
      LD      M404  ; 各個実行
      AND     Y1142
      OR      M300  ; 原点復帰PB
      ANI     L103
      ORB
      LD      M675
      LD      M419  ; 初期SOL励磁
      AND     M325
      ORB
      ANI     M674
      ORB
      AND     M17  ; 運転ﾓｰﾄﾞ切替
      AND     X0  ; 運転準備入り
      OUT     M675
1935  LD      M675
      ANI     Y30A
      OUT     Y309
1938  LD      M674
      ANI     Y309
      OUT     Y30A
1941  LD      M421  ; 連続運転
      AND     T198
      ANI     L102
      AND     M322
      AND     M325
      AND     M17  ; 運転ﾓｰﾄﾞ切替
      AND     X0  ; 運転準備入り
      OUT     M676
1949  LD      M421  ; 連続運転
      AND     M676
      FMOVP   K0 D1520 K2
      MPS
      LD      SM412  ; 1秒 ｸﾛｯｸ
      OR      M1300
      ANB
      ANI     M1301
      ANI     M1303
      OUT     M1300
      AND     SM412  ; 1秒 ｸﾛｯｸ
      INCP    D1520
      MRD
      ANI     M1303
      AND<    D1500 D1520
      OUT     M1301
      AND     SM412  ; 1秒 ｸﾛｯｸ
      INCP    D1521
      MPP
      AND<    D1501 D1521
      OUT     M1303
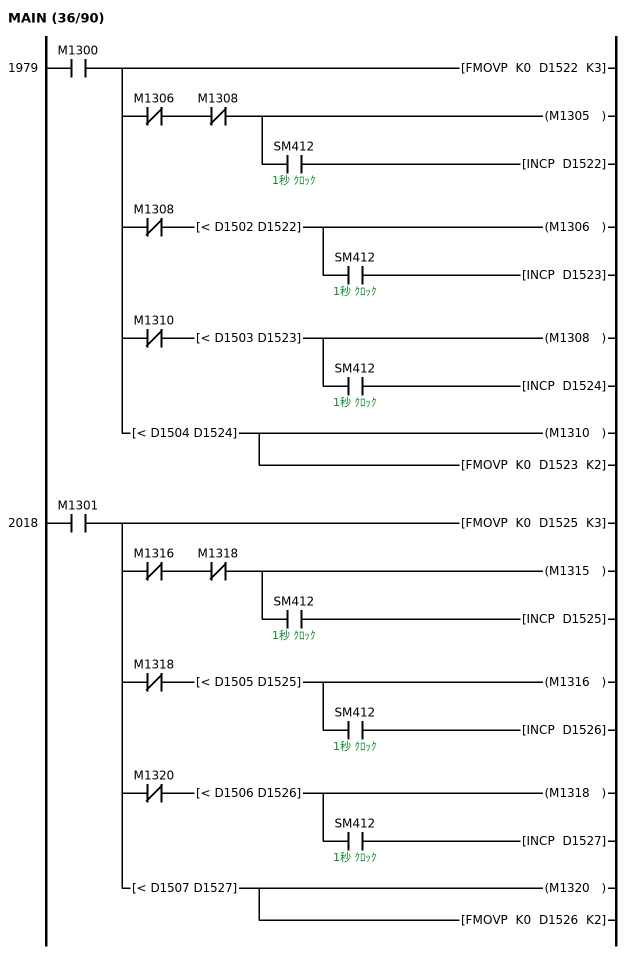
1979  LD      M1300
      FMOVP   K0 D1522 K3
      MPS
      ANI     M1306
      ANI     M1308
      OUT     M1305
      AND     SM412  ; 1秒 ｸﾛｯｸ
      INCP    D1522
      MRD
      ANI     M1308
      AND<    D1502 D1522
      OUT     M1306
      AND     SM412  ; 1秒 ｸﾛｯｸ
      INCP    D1523
      MRD
      ANI     M1310
      AND<    D1503 D1523
      OUT     M1308
      AND     SM412  ; 1秒 ｸﾛｯｸ
      INCP    D1524
      MPP
      AND<    D1504 D1524
      OUT     M1310
      FMOVP   K0 D1523 K2
2018  LD      M1301
      FMOVP   K0 D1525 K3
      MPS
      ANI     M1316
      ANI     M1318
      OUT     M1315
      AND     SM412  ; 1秒 ｸﾛｯｸ
      INCP    D1525
      MRD
      ANI     M1318
      AND<    D1505 D1525
      OUT     M1316
      AND     SM412  ; 1秒 ｸﾛｯｸ
      INCP    D1526
      MRD
      ANI     M1320
      AND<    D1506 D1526
      OUT     M1318
      AND     SM412  ; 1秒 ｸﾛｯｸ
      INCP    D1527
      MPP
      AND<    D1507 D1527
      OUT     M1320
      FMOVP   K0 D1526 K2
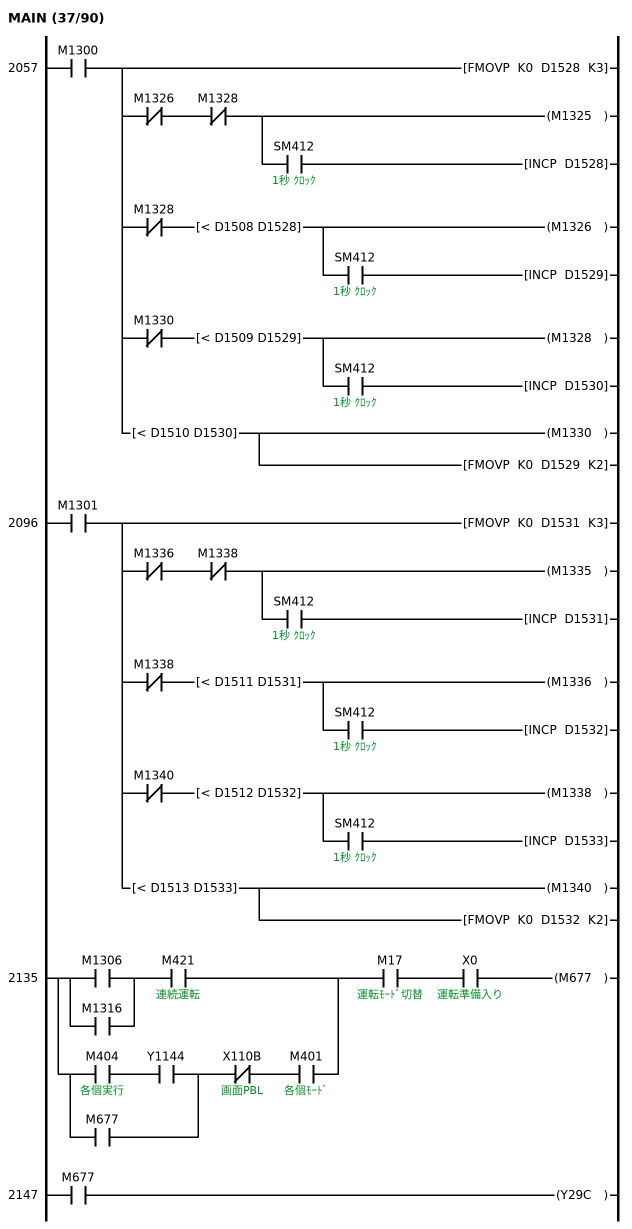
2057  LD      M1300
      FMOVP   K0 D1528 K3
      MPS
      ANI     M1326
      ANI     M1328
      OUT     M1325
      AND     SM412  ; 1秒 ｸﾛｯｸ
      INCP    D1528
      MRD
      ANI     M1328
      AND<    D1508 D1528
      OUT     M1326
      AND     SM412  ; 1秒 ｸﾛｯｸ
      INCP    D1529
      MRD
      ANI     M1330
      AND<    D1509 D1529
      OUT     M1328
      AND     SM412  ; 1秒 ｸﾛｯｸ
      INCP    D1530
      MPP
      AND<    D1510 D1530
      OUT     M1330
      FMOVP   K0 D1529 K2
2096  LD      M1301
      FMOVP   K0 D1531 K3
      MPS
      ANI     M1336
      ANI     M1338
      OUT     M1335
      AND     SM412  ; 1秒 ｸﾛｯｸ
      INCP    D1531
      MRD
      ANI     M1338
      AND<    D1511 D1531
      OUT     M1336
      AND     SM412  ; 1秒 ｸﾛｯｸ
      INCP    D1532
      MRD
      ANI     M1340
      AND<    D1512 D1532
      OUT     M1338
      AND     SM412  ; 1秒 ｸﾛｯｸ
      INCP    D1533
      MPP
      AND<    D1513 D1533
      OUT     M1340
      FMOVP   K0 D1532 K2
2135  LD      M1306
      OR      M1316
      AND     M421  ; 連続運転
      LD      M404  ; 各個実行
      AND     Y1144
      OR      M677
      ANI     X110B  ; 画面PBL
      AND     M401  ; 各個ﾓｰﾄﾞ
      ORB
      AND     M17  ; 運転ﾓｰﾄﾞ切替
      AND     X0  ; 運転準備入り
      OUT     M677
2147  LD      M677
      OUT     Y29C
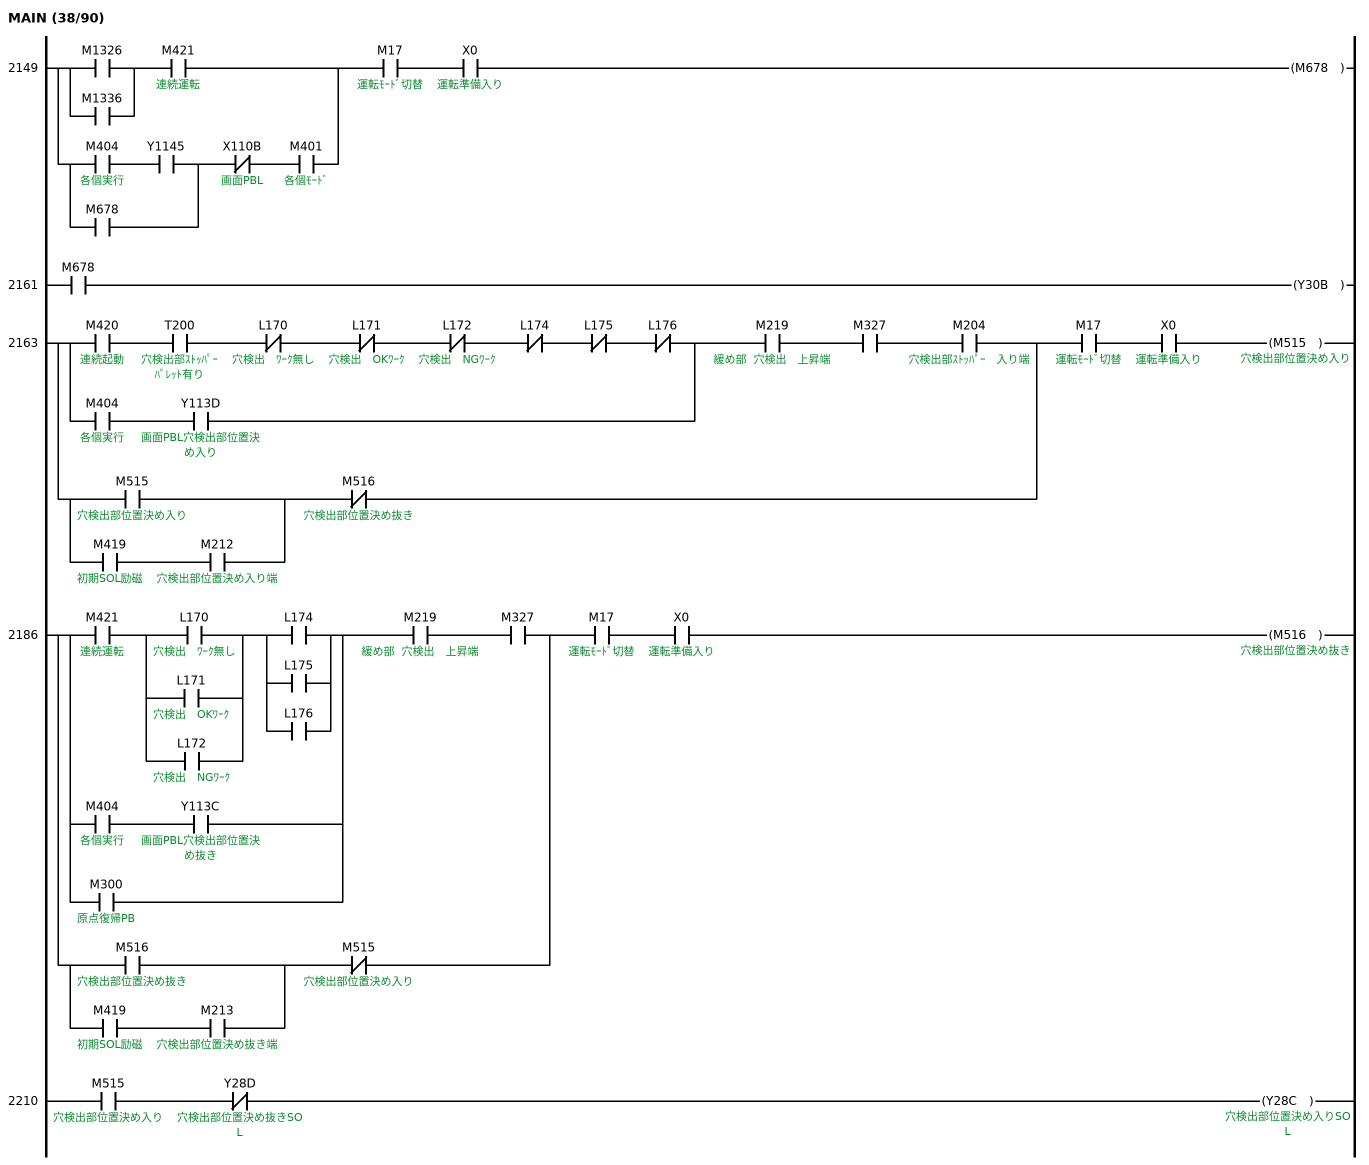
2149  LD      M1326
      OR      M1336
      AND     M421  ; 連続運転
      LD      M404  ; 各個実行
      AND     Y1145
      OR      M678
      ANI     X110B  ; 画面PBL
      AND     M401  ; 各個ﾓｰﾄﾞ
      ORB
      AND     M17  ; 運転ﾓｰﾄﾞ切替
      AND     X0  ; 運転準備入り
      OUT     M678
2161  LD      M678
      OUT     Y30B
2163  LD      M420  ; 連続起動
      AND     T200  ; 穴検出部ｽﾄｯﾊﾟｰ 　ﾊﾟﾚｯﾄ有り
      ANI     L170  ; 穴検出　ﾜｰｸ無し
      ANI     L171  ; 穴検出　OKﾜｰｸ
      ANI     L172  ; 穴検出　NGﾜｰｸ
      ANI     L174
      ANI     L175
      ANI     L176
      LD      M404  ; 各個実行
      AND     Y113D  ; 画面PBL穴検出部位置決め入り
      ORB
      AND     M219  ; 緩め部  穴検出　上昇端
      AND     M327
      AND     M204  ; 穴検出部ｽﾄｯﾊﾟｰ　入り端
      LD      M515  ; 穴検出部位置決め入り
      LD      M419  ; 初期SOL励磁
      AND     M212  ; 穴検出部位置決め入り端
      ORB
      ANI     M516  ; 穴検出部位置決め抜き
      ORB
      AND     M17  ; 運転ﾓｰﾄﾞ切替
      AND     X0  ; 運転準備入り
      OUT     M515  ; 穴検出部位置決め入り
2186  LD      M421  ; 連続運転
      LD      L170  ; 穴検出　ﾜｰｸ無し
      OR      L171  ; 穴検出　OKﾜｰｸ
      OR      L172  ; 穴検出　NGﾜｰｸ
      ANB
      LD      L174
      OR      L175
      OR      L176
      ANB
      LD      M404  ; 各個実行
      AND     Y113C  ; 画面PBL穴検出部位置決め抜き
      ORB
      OR      M300  ; 原点復帰PB
      AND     M219  ; 緩め部  穴検出　上昇端
      AND     M327
      LD      M516  ; 穴検出部位置決め抜き
      LD      M419  ; 初期SOL励磁
      AND     M213  ; 穴検出部位置決め抜き端
      ORB
      ANI     M515  ; 穴検出部位置決め入り
      ORB
      AND     M17  ; 運転ﾓｰﾄﾞ切替
      AND     X0  ; 運転準備入り
      OUT     M516  ; 穴検出部位置決め抜き
2210  LD      M515  ; 穴検出部位置決め入り
      ANI     Y28D  ; 穴検出部位置決め抜きSOL
      OUT     Y28C  ; 穴検出部位置決め入りSOL
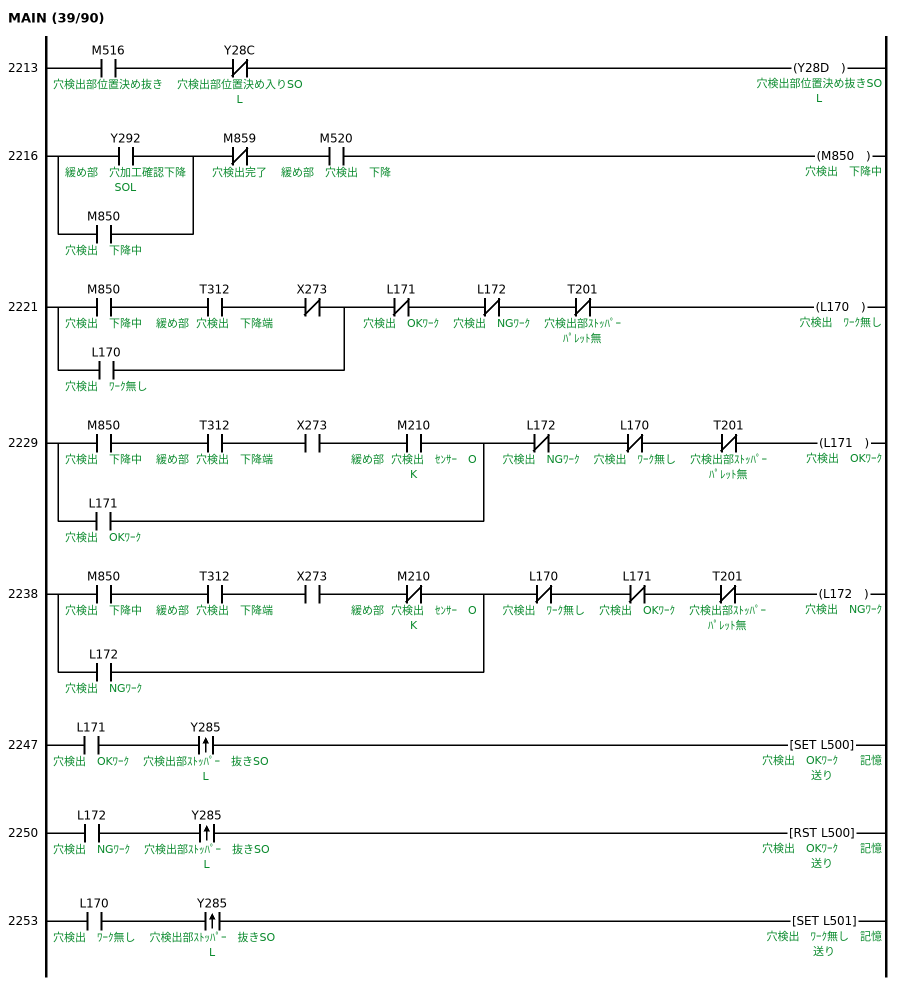
2213  LD      M516  ; 穴検出部位置決め抜き
      ANI     Y28C  ; 穴検出部位置決め入りSOL
      OUT     Y28D  ; 穴検出部位置決め抜きSOL
2216  LD      Y292  ; 緩め部　穴加工確認下降 SOL
      OR      M850  ; 穴検出　下降中
      ANI     M859  ; 穴検出完了
      AND     M520  ; 緩め部　穴検出　下降
      OUT     M850  ; 穴検出　下降中
2221  LD      M850  ; 穴検出　下降中
      AND     T312  ; 緩め部  穴検出　下降端
      ANI     X273
      OR      L170  ; 穴検出　ﾜｰｸ無し
      ANI     L171  ; 穴検出　OKﾜｰｸ
      ANI     L172  ; 穴検出　NGﾜｰｸ
      ANI     T201  ; 穴検出部ｽﾄｯﾊﾟｰ 　ﾊﾟﾚｯﾄ無
      OUT     L170  ; 穴検出　ﾜｰｸ無し
2229  LD      M850  ; 穴検出　下降中
      AND     T312  ; 緩め部  穴検出　下降端
      AND     X273
      AND     M210  ; 緩め部  穴検出　ｾﾝｻｰ　OK
      OR      L171  ; 穴検出　OKﾜｰｸ
      ANI     L172  ; 穴検出　NGﾜｰｸ
      ANI     L170  ; 穴検出　ﾜｰｸ無し
      ANI     T201  ; 穴検出部ｽﾄｯﾊﾟｰ 　ﾊﾟﾚｯﾄ無
      OUT     L171  ; 穴検出　OKﾜｰｸ
2238  LD      M850  ; 穴検出　下降中
      AND     T312  ; 緩め部  穴検出　下降端
      AND     X273
      ANI     M210  ; 緩め部  穴検出　ｾﾝｻｰ　OK
      OR      L172  ; 穴検出　NGﾜｰｸ
      ANI     L170  ; 穴検出　ﾜｰｸ無し
      ANI     L171  ; 穴検出　OKﾜｰｸ
      ANI     T201  ; 穴検出部ｽﾄｯﾊﾟｰ 　ﾊﾟﾚｯﾄ無
      OUT     L172  ; 穴検出　NGﾜｰｸ
2247  LD      L171  ; 穴検出　OKﾜｰｸ
      ANDP    Y285  ; 穴検出部ｽﾄｯﾊﾟｰ　抜きSOL
      SET     L500  ; 穴検出　OKﾜｰｸ　　記憶送り
2250  LD      L172  ; 穴検出　NGﾜｰｸ
      ANDP    Y285  ; 穴検出部ｽﾄｯﾊﾟｰ　抜きSOL
      RST     L500  ; 穴検出　OKﾜｰｸ　　記憶送り
2253  LD      L170  ; 穴検出　ﾜｰｸ無し
      ANDP    Y285  ; 穴検出部ｽﾄｯﾊﾟｰ　抜きSOL
      SET     L501  ; 穴検出　ﾜｰｸ無し　記憶送り
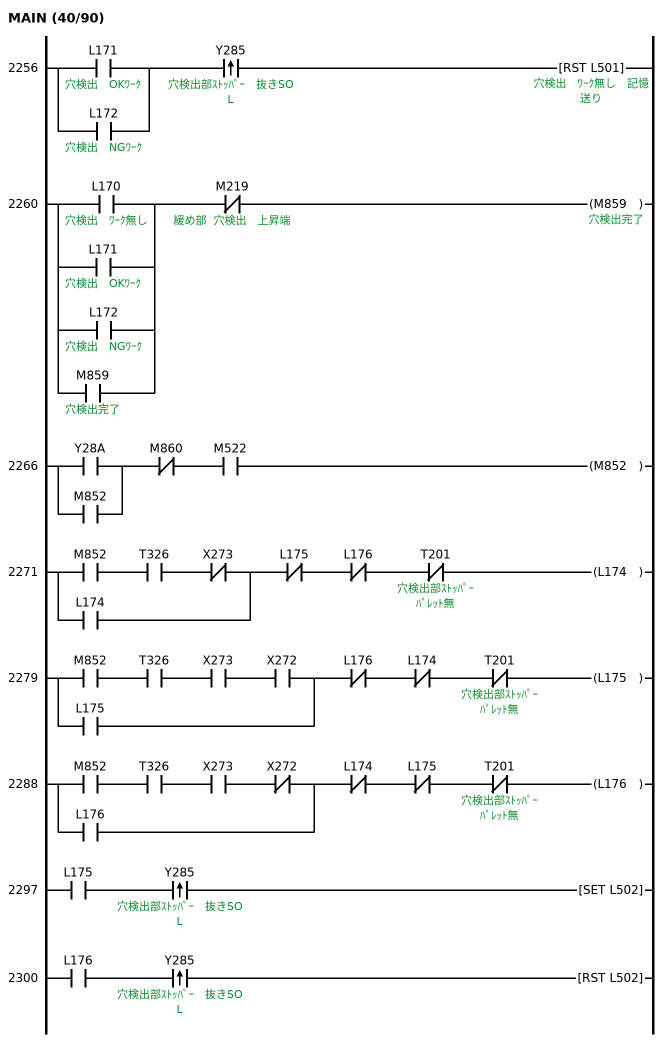
2256  LD      L171  ; 穴検出　OKﾜｰｸ
      OR      L172  ; 穴検出　NGﾜｰｸ
      ANDP    Y285  ; 穴検出部ｽﾄｯﾊﾟｰ　抜きSOL
      RST     L501  ; 穴検出　ﾜｰｸ無し　記憶送り
2260  LD      L170  ; 穴検出　ﾜｰｸ無し
      OR      L171  ; 穴検出　OKﾜｰｸ
      OR      L172  ; 穴検出　NGﾜｰｸ
      OR      M859  ; 穴検出完了
      ANI     M219  ; 緩め部  穴検出　上昇端
      OUT     M859  ; 穴検出完了
2266  LD      Y28A
      OR      M852
      ANI     M860
      AND     M522
      OUT     M852
2271  LD      M852
      AND     T326
      ANI     X273
      OR      L174
      ANI     L175
      ANI     L176
      ANI     T201  ; 穴検出部ｽﾄｯﾊﾟｰ 　ﾊﾟﾚｯﾄ無
      OUT     L174
2279  LD      M852
      AND     T326
      AND     X273
      AND     X272
      OR      L175
      ANI     L176
      ANI     L174
      ANI     T201  ; 穴検出部ｽﾄｯﾊﾟｰ 　ﾊﾟﾚｯﾄ無
      OUT     L175
2288  LD      M852
      AND     T326
      AND     X273
      ANI     X272
      OR      L176
      ANI     L174
      ANI     L175
      ANI     T201  ; 穴検出部ｽﾄｯﾊﾟｰ 　ﾊﾟﾚｯﾄ無
      OUT     L176
2297  LD      L175
      ANDP    Y285  ; 穴検出部ｽﾄｯﾊﾟｰ　抜きSOL
      SET     L502
2300  LD      L176
      ANDP    Y285  ; 穴検出部ｽﾄｯﾊﾟｰ　抜きSOL
      RST     L502
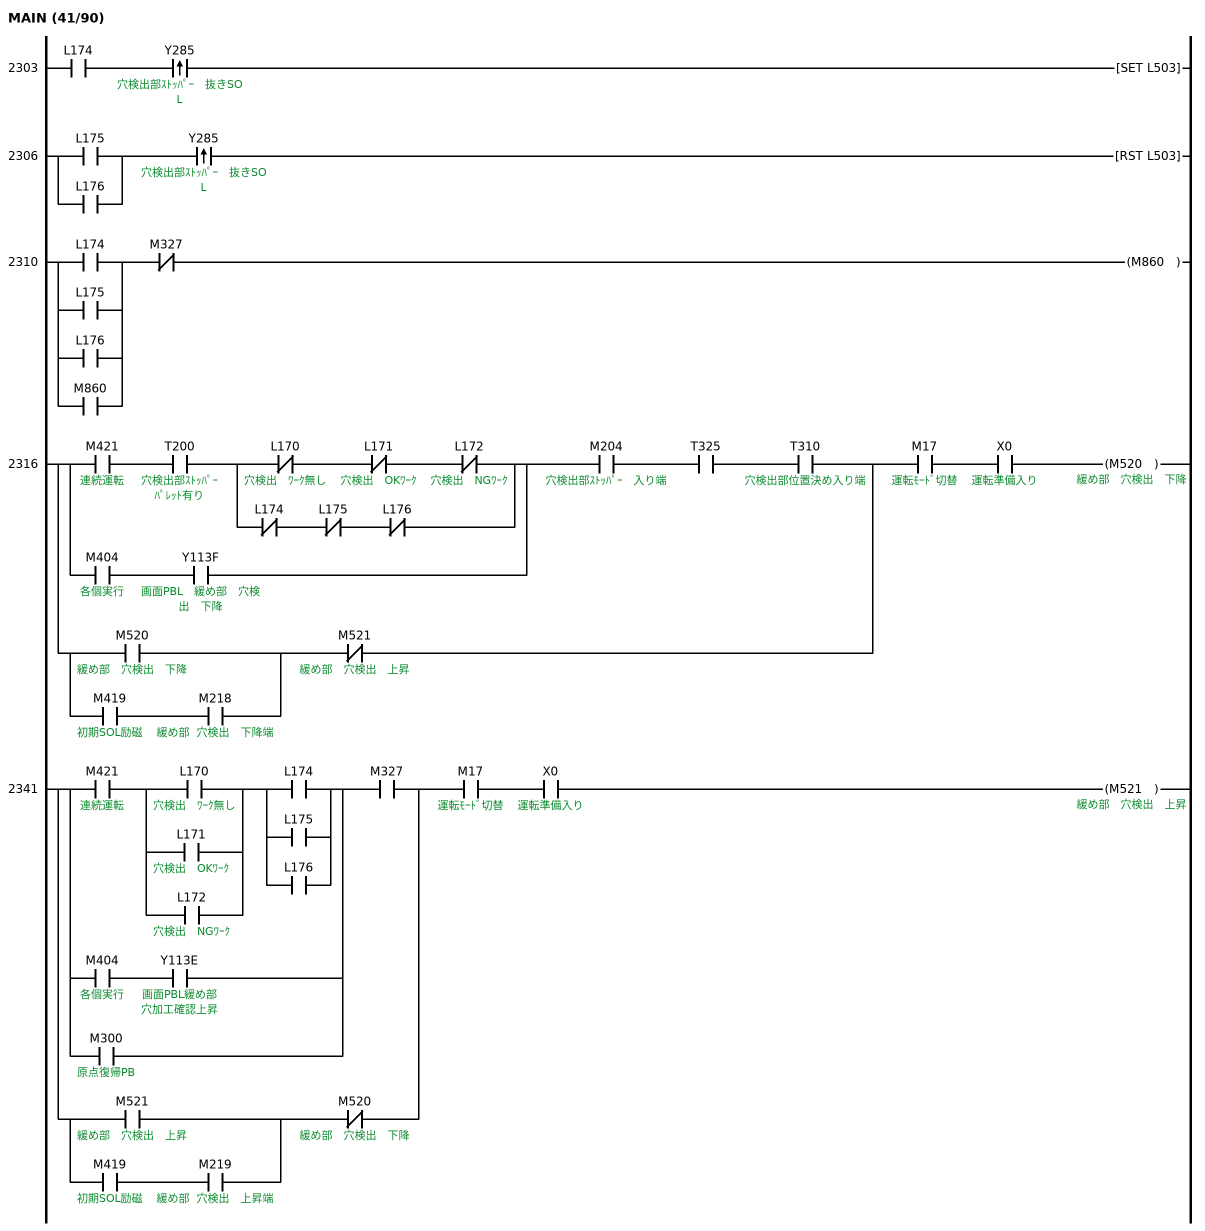
2303  LD      L174
      ANDP    Y285  ; 穴検出部ｽﾄｯﾊﾟｰ　抜きSOL
      SET     L503
2306  LD      L175
      OR      L176
      ANDP    Y285  ; 穴検出部ｽﾄｯﾊﾟｰ　抜きSOL
      RST     L503
2310  LD      L174
      OR      L175
      OR      L176
      OR      M860
      ANI     M327
      OUT     M860
2316  LD      M421  ; 連続運転
      AND     T200  ; 穴検出部ｽﾄｯﾊﾟｰ 　ﾊﾟﾚｯﾄ有り
      LDI     L170  ; 穴検出　ﾜｰｸ無し
      ANI     L171  ; 穴検出　OKﾜｰｸ
      ANI     L172  ; 穴検出　NGﾜｰｸ
      LDI     L174
      ANI     L175
      ANI     L176
      ORB
      ANB
      LD      M404  ; 各個実行
      AND     Y113F  ; 画面PBL　緩め部　穴検出　下降
      ORB
      AND     M204  ; 穴検出部ｽﾄｯﾊﾟｰ　入り端
      AND     T325
      AND     T310  ; 穴検出部位置決め入り端
      LD      M520  ; 緩め部　穴検出　下降
      LD      M419  ; 初期SOL励磁
      AND     M218  ; 緩め部  穴検出　下降端
      ORB
      ANI     M521  ; 緩め部　穴検出　上昇
      ORB
      AND     M17  ; 運転ﾓｰﾄﾞ切替
      AND     X0  ; 運転準備入り
      OUT     M520  ; 緩め部　穴検出　下降
2341  LD      M421  ; 連続運転
      LD      L170  ; 穴検出　ﾜｰｸ無し
      OR      L171  ; 穴検出　OKﾜｰｸ
      OR      L172  ; 穴検出　NGﾜｰｸ
      ANB
      LD      L174
      OR      L175
      OR      L176
      ANB
      LD      M404  ; 各個実行
      AND     Y113E  ; 画面PBL緩め部 穴加工確認上昇
      ORB
      OR      M300  ; 原点復帰PB
      AND     M327
      LD      M521  ; 緩め部　穴検出　上昇
      LD      M419  ; 初期SOL励磁
      AND     M219  ; 緩め部  穴検出　上昇端
      ORB
      ANI     M520  ; 緩め部　穴検出　下降
      ORB
      AND     M17  ; 運転ﾓｰﾄﾞ切替
      AND     X0  ; 運転準備入り
      OUT     M521  ; 緩め部　穴検出　上昇
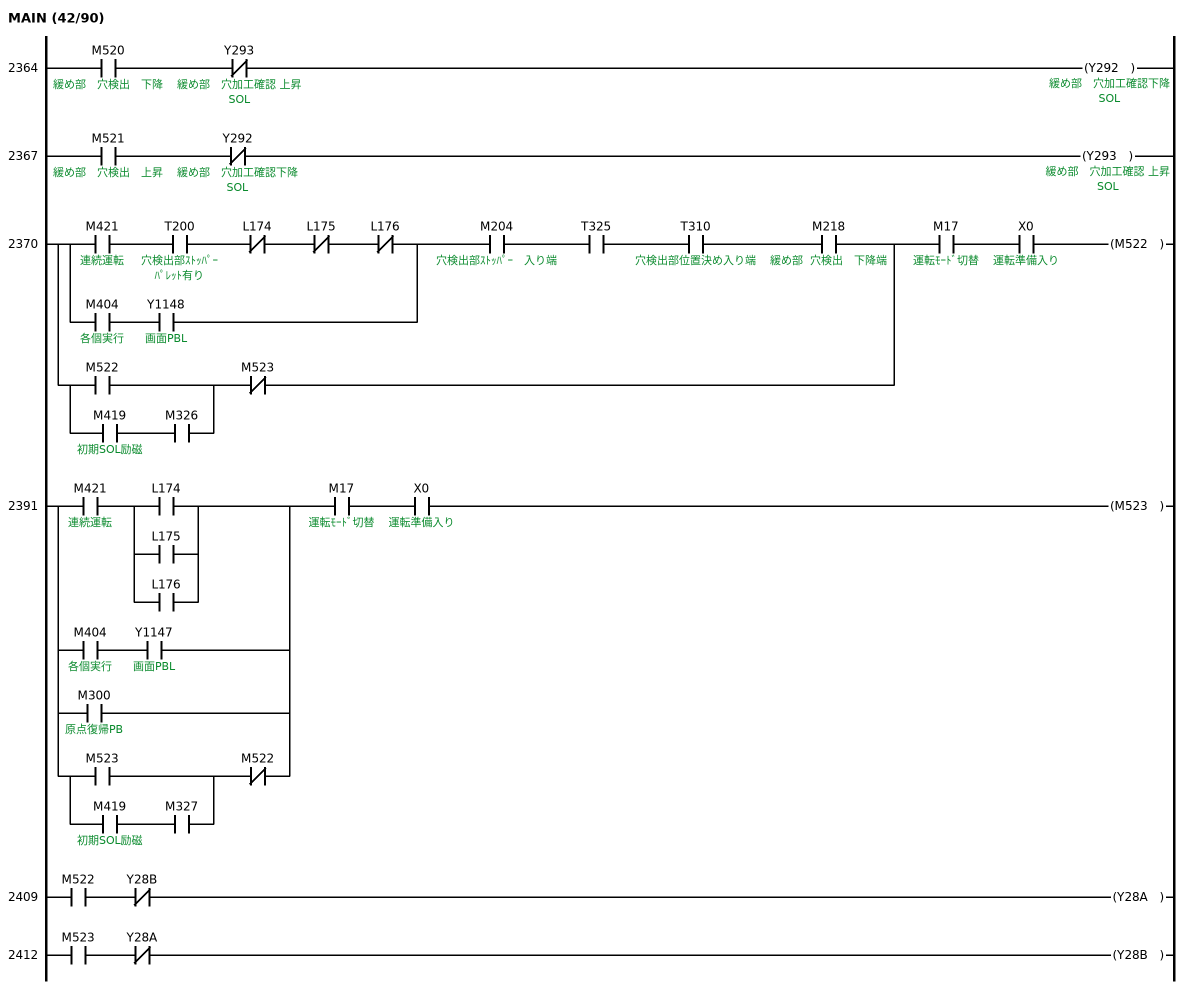
2364  LD      M520  ; 緩め部　穴検出　下降
      ANI     Y293  ; 緩め部　穴加工確認 上昇 SOL
      OUT     Y292  ; 緩め部　穴加工確認下降 SOL
2367  LD      M521  ; 緩め部　穴検出　上昇
      ANI     Y292  ; 緩め部　穴加工確認下降 SOL
      OUT     Y293  ; 緩め部　穴加工確認 上昇 SOL
2370  LD      M421  ; 連続運転
      AND     T200  ; 穴検出部ｽﾄｯﾊﾟｰ 　ﾊﾟﾚｯﾄ有り
      ANI     L174
      ANI     L175
      ANI     L176
      LD      M404  ; 各個実行
      AND     Y1148  ; 画面PBL
      ORB
      AND     M204  ; 穴検出部ｽﾄｯﾊﾟｰ　入り端
      AND     T325
      AND     T310  ; 穴検出部位置決め入り端
      AND     M218  ; 緩め部  穴検出　下降端
      LD      M522
      LD      M419  ; 初期SOL励磁
      AND     M326
      ORB
      ANI     M523
      ORB
      AND     M17  ; 運転ﾓｰﾄﾞ切替
      AND     X0  ; 運転準備入り
      OUT     M522
2391  LD      M421  ; 連続運転
      LD      L174
      OR      L175
      OR      L176
      ANB
      LD      M404  ; 各個実行
      AND     Y1147  ; 画面PBL
      ORB
      OR      M300  ; 原点復帰PB
      LD      M523
      LD      M419  ; 初期SOL励磁
      AND     M327
      ORB
      ANI     M522
      ORB
      AND     M17  ; 運転ﾓｰﾄﾞ切替
      AND     X0  ; 運転準備入り
      OUT     M523
2409  LD      M522
      ANI     Y28B
      OUT     Y28A
2412  LD      M523
      ANI     Y28A
      OUT     Y28B
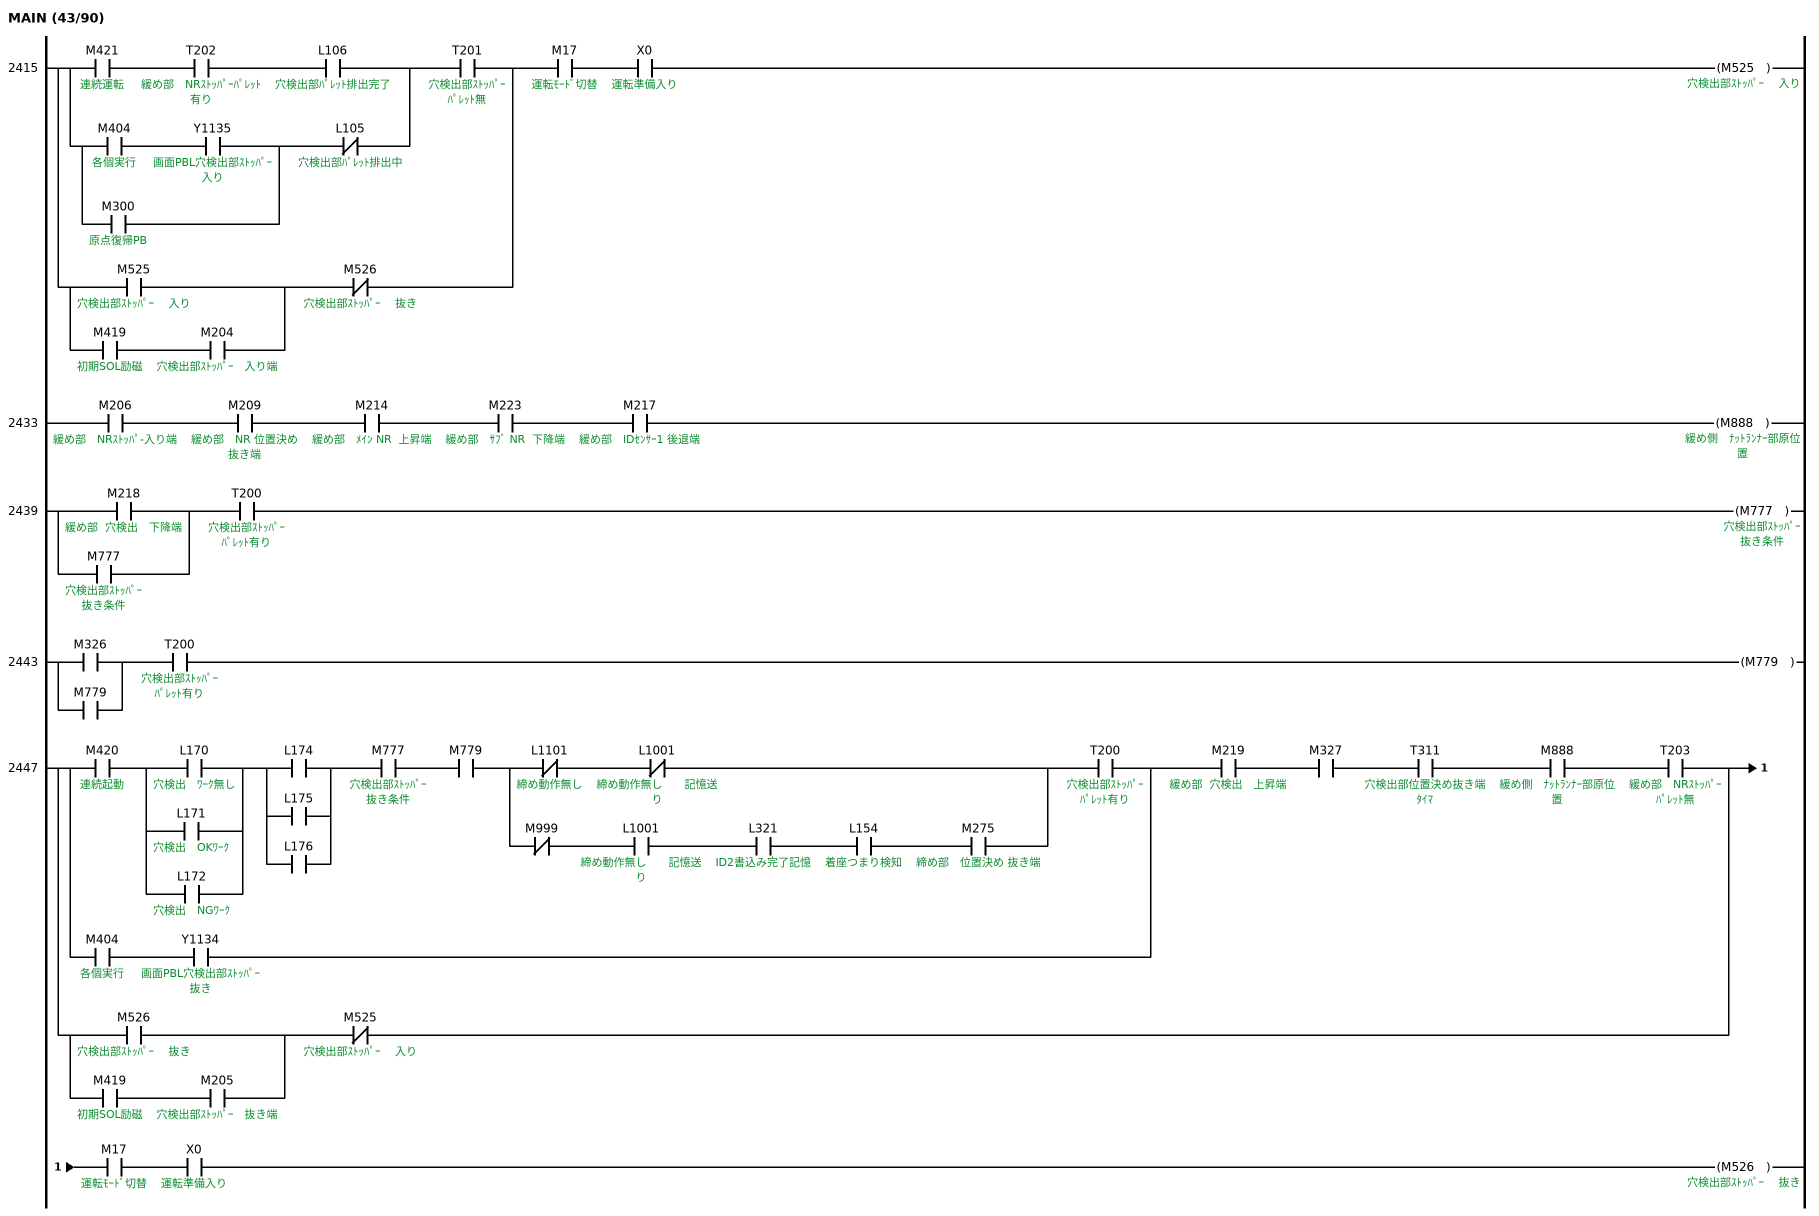
2415  LD      M421  ; 連続運転
      AND     T202  ; 緩め部　NRｽﾄｯﾊﾟｰﾊﾟﾚｯﾄ有り
      AND     L106  ; 穴検出部ﾊﾟﾚｯﾄ排出完了
      LD      M404  ; 各個実行
      AND     Y1135  ; 画面PBL穴検出部ｽﾄｯﾊﾟｰ 　入り
      OR      M300  ; 原点復帰PB
      ANI     L105  ; 穴検出部ﾊﾟﾚｯﾄ排出中
      ORB
      AND     T201  ; 穴検出部ｽﾄｯﾊﾟｰ 　ﾊﾟﾚｯﾄ無
      LD      M525  ; 穴検出部ｽﾄｯﾊﾟｰ 　入り
      LD      M419  ; 初期SOL励磁
      AND     M204  ; 穴検出部ｽﾄｯﾊﾟｰ　入り端
      ORB
      ANI     M526  ; 穴検出部ｽﾄｯﾊﾟｰ 　抜き
      ORB
      AND     M17  ; 運転ﾓｰﾄﾞ切替
      AND     X0  ; 運転準備入り
      OUT     M525  ; 穴検出部ｽﾄｯﾊﾟｰ 　入り
2433  LD      M206  ; 緩め部　NRｽﾄｯﾊﾟ-入り端
      AND     M209  ; 緩め部　NR 位置決め 抜き端
      AND     M214  ; 緩め部　ﾒｲﾝ NR  上昇端
      AND     M223  ; 緩め部　ｻﾌﾞ NR  下降端
      AND     M217  ; 緩め部　IDｾﾝｻｰ1 後退端
      OUT     M888  ; 緩め側　ﾅｯﾄﾗﾝﾅｰ部原位置
2439  LD      M218  ; 緩め部  穴検出　下降端
      OR      M777  ; 穴検出部ｽﾄｯﾊﾟｰ 　抜き条件
      AND     T200  ; 穴検出部ｽﾄｯﾊﾟｰ 　ﾊﾟﾚｯﾄ有り
      OUT     M777  ; 穴検出部ｽﾄｯﾊﾟｰ 　抜き条件
2443  LD      M326
      OR      M779
      AND     T200  ; 穴検出部ｽﾄｯﾊﾟｰ 　ﾊﾟﾚｯﾄ有り
      OUT     M779
2447  LD      M420  ; 連続起動
      LD      L170  ; 穴検出　ﾜｰｸ無し
      OR      L171  ; 穴検出　OKﾜｰｸ
      OR      L172  ; 穴検出　NGﾜｰｸ
      ANB
      LD      L174
      OR      L175
      OR      L176
      ANB
      AND     M777  ; 穴検出部ｽﾄｯﾊﾟｰ 　抜き条件
      AND     M779
      LDI     L1101  ; 締め動作無し
      ANI     L1001  ; 締め動作無し　　記憶送り
      LDI     M999
      AND     L1001  ; 締め動作無し　　記憶送り
      AND     L321  ; ID2書込み完了記憶
      AND     L154  ; 着座つまり検知
      AND     M275  ; 締め部　位置決め 抜き端
      ORB
      ANB
      AND     T200  ; 穴検出部ｽﾄｯﾊﾟｰ 　ﾊﾟﾚｯﾄ有り
      LD      M404  ; 各個実行
      AND     Y1134  ; 画面PBL穴検出部ｽﾄｯﾊﾟｰ 　抜き
      ORB
      AND     M219  ; 緩め部  穴検出　上昇端
      AND     M327
      AND     T311  ; 穴検出部位置決め抜き端　ﾀｲﾏ
      AND     M888  ; 緩め側　ﾅｯﾄﾗﾝﾅｰ部原位置
      AND     T203  ; 緩め部　NRｽﾄｯﾊﾟｰ ﾊﾟﾚｯﾄ無
      LD      M526  ; 穴検出部ｽﾄｯﾊﾟｰ 　抜き
      LD      M419  ; 初期SOL励磁
      AND     M205  ; 穴検出部ｽﾄｯﾊﾟｰ　抜き端
      ORB
      ANI     M525  ; 穴検出部ｽﾄｯﾊﾟｰ 　入り
      ORB
      AND     M17  ; 運転ﾓｰﾄﾞ切替
      AND     X0  ; 運転準備入り
      OUT     M526  ; 穴検出部ｽﾄｯﾊﾟｰ 　抜き
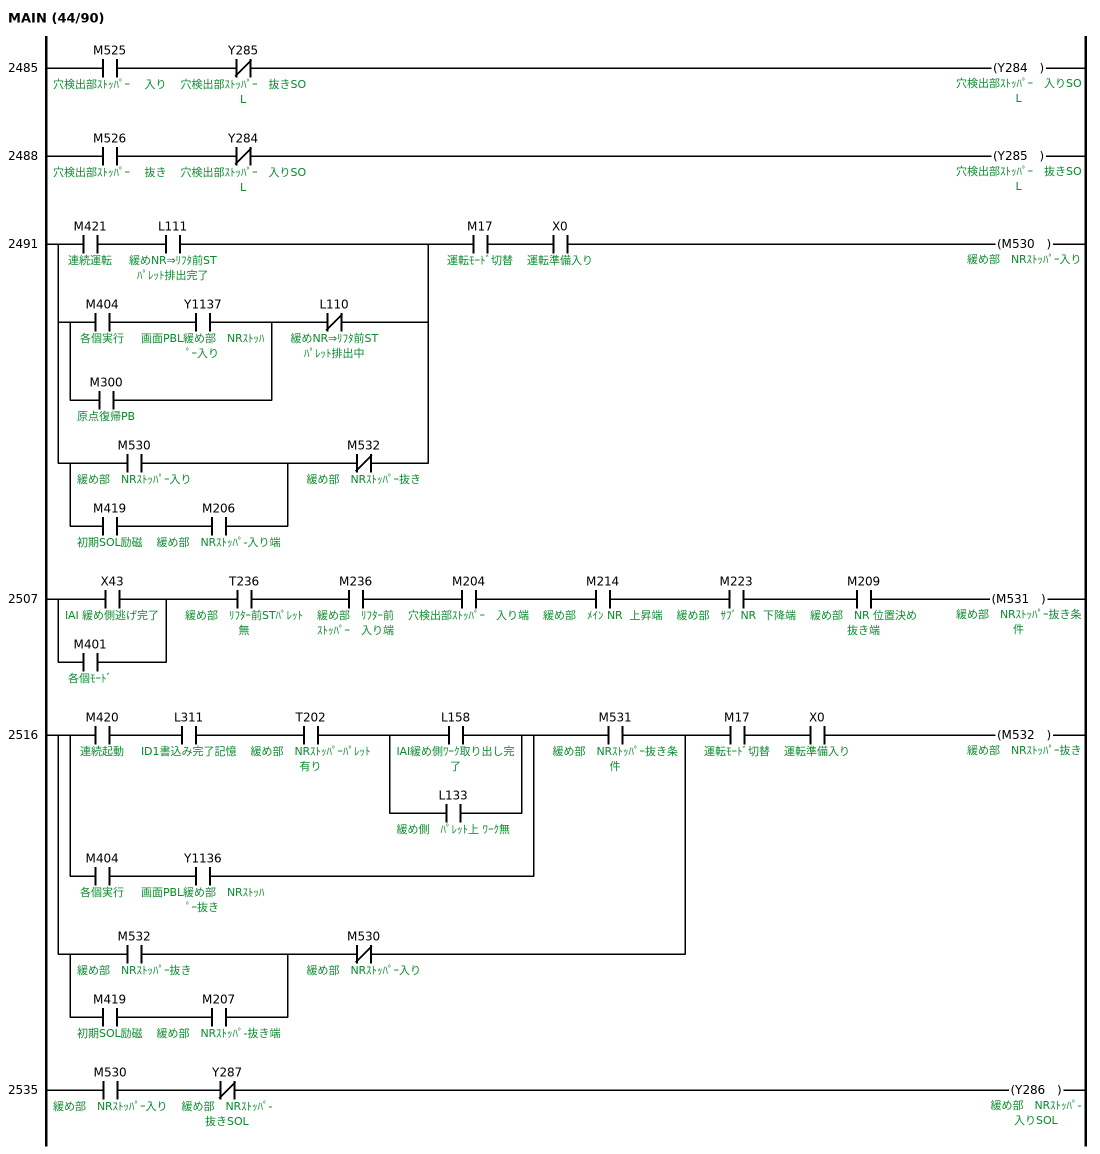
2485  LD      M525  ; 穴検出部ｽﾄｯﾊﾟｰ 　入り
      ANI     Y285  ; 穴検出部ｽﾄｯﾊﾟｰ　抜きSOL
      OUT     Y284  ; 穴検出部ｽﾄｯﾊﾟｰ　入りSOL
2488  LD      M526  ; 穴検出部ｽﾄｯﾊﾟｰ 　抜き
      ANI     Y284  ; 穴検出部ｽﾄｯﾊﾟｰ　入りSOL
      OUT     Y285  ; 穴検出部ｽﾄｯﾊﾟｰ　抜きSOL
2491  LD      M421  ; 連続運転
      AND     L111  ; 緩めNR⇒ﾘﾌﾀ前ST ﾊﾟﾚｯﾄ排出完了
      LD      M404  ; 各個実行
      AND     Y1137  ; 画面PBL緩め部　NRｽﾄｯﾊﾟｰ入り
      OR      M300  ; 原点復帰PB
      ANI     L110  ; 緩めNR⇒ﾘﾌﾀ前ST ﾊﾟﾚｯﾄ排出中
      ORB
      LD      M530  ; 緩め部　NRｽﾄｯﾊﾟｰ入り
      LD      M419  ; 初期SOL励磁
      AND     M206  ; 緩め部　NRｽﾄｯﾊﾟ-入り端
      ORB
      ANI     M532  ; 緩め部　NRｽﾄｯﾊﾟｰ抜き
      ORB
      AND     M17  ; 運転ﾓｰﾄﾞ切替
      AND     X0  ; 運転準備入り
      OUT     M530  ; 緩め部　NRｽﾄｯﾊﾟｰ入り
2507  LD      X43  ; IAI 緩め側逃げ完了
      OR      M401  ; 各個ﾓｰﾄﾞ
      AND     T236  ; 緩め部　ﾘﾌﾀｰ前STﾊﾟﾚｯﾄ無
      AND     M236  ; 緩め部　ﾘﾌﾀｰ前  ｽﾄｯﾊﾟｰ　入り端
      AND     M204  ; 穴検出部ｽﾄｯﾊﾟｰ　入り端
      AND     M214  ; 緩め部　ﾒｲﾝ NR  上昇端
      AND     M223  ; 緩め部　ｻﾌﾞ NR  下降端
      AND     M209  ; 緩め部　NR 位置決め 抜き端
      OUT     M531  ; 緩め部　NRｽﾄｯﾊﾟｰ抜き条件
2516  LD      M420  ; 連続起動
      AND     L311  ; ID1書込み完了記憶
      AND     T202  ; 緩め部　NRｽﾄｯﾊﾟｰﾊﾟﾚｯﾄ有り
      LD      L158  ; IAI緩め側ﾜｰｸ取り出し完了
      OR      L133  ; 緩め側　ﾊﾟﾚｯﾄ上 ﾜｰｸ無
      ANB
      LD      M404  ; 各個実行
      AND     Y1136  ; 画面PBL緩め部　NRｽﾄｯﾊﾟｰ抜き
      ORB
      AND     M531  ; 緩め部　NRｽﾄｯﾊﾟｰ抜き条件
      LD      M532  ; 緩め部　NRｽﾄｯﾊﾟｰ抜き
      LD      M419  ; 初期SOL励磁
      AND     M207  ; 緩め部　NRｽﾄｯﾊﾟ-抜き端
      ORB
      ANI     M530  ; 緩め部　NRｽﾄｯﾊﾟｰ入り
      ORB
      AND     M17  ; 運転ﾓｰﾄﾞ切替
      AND     X0  ; 運転準備入り
      OUT     M532  ; 緩め部　NRｽﾄｯﾊﾟｰ抜き
2535  LD      M530  ; 緩め部　NRｽﾄｯﾊﾟｰ入り
      ANI     Y287  ; 緩め部　NRｽﾄｯﾊﾟ-抜きSOL
      OUT     Y286  ; 緩め部　NRｽﾄｯﾊﾟ-入りSOL
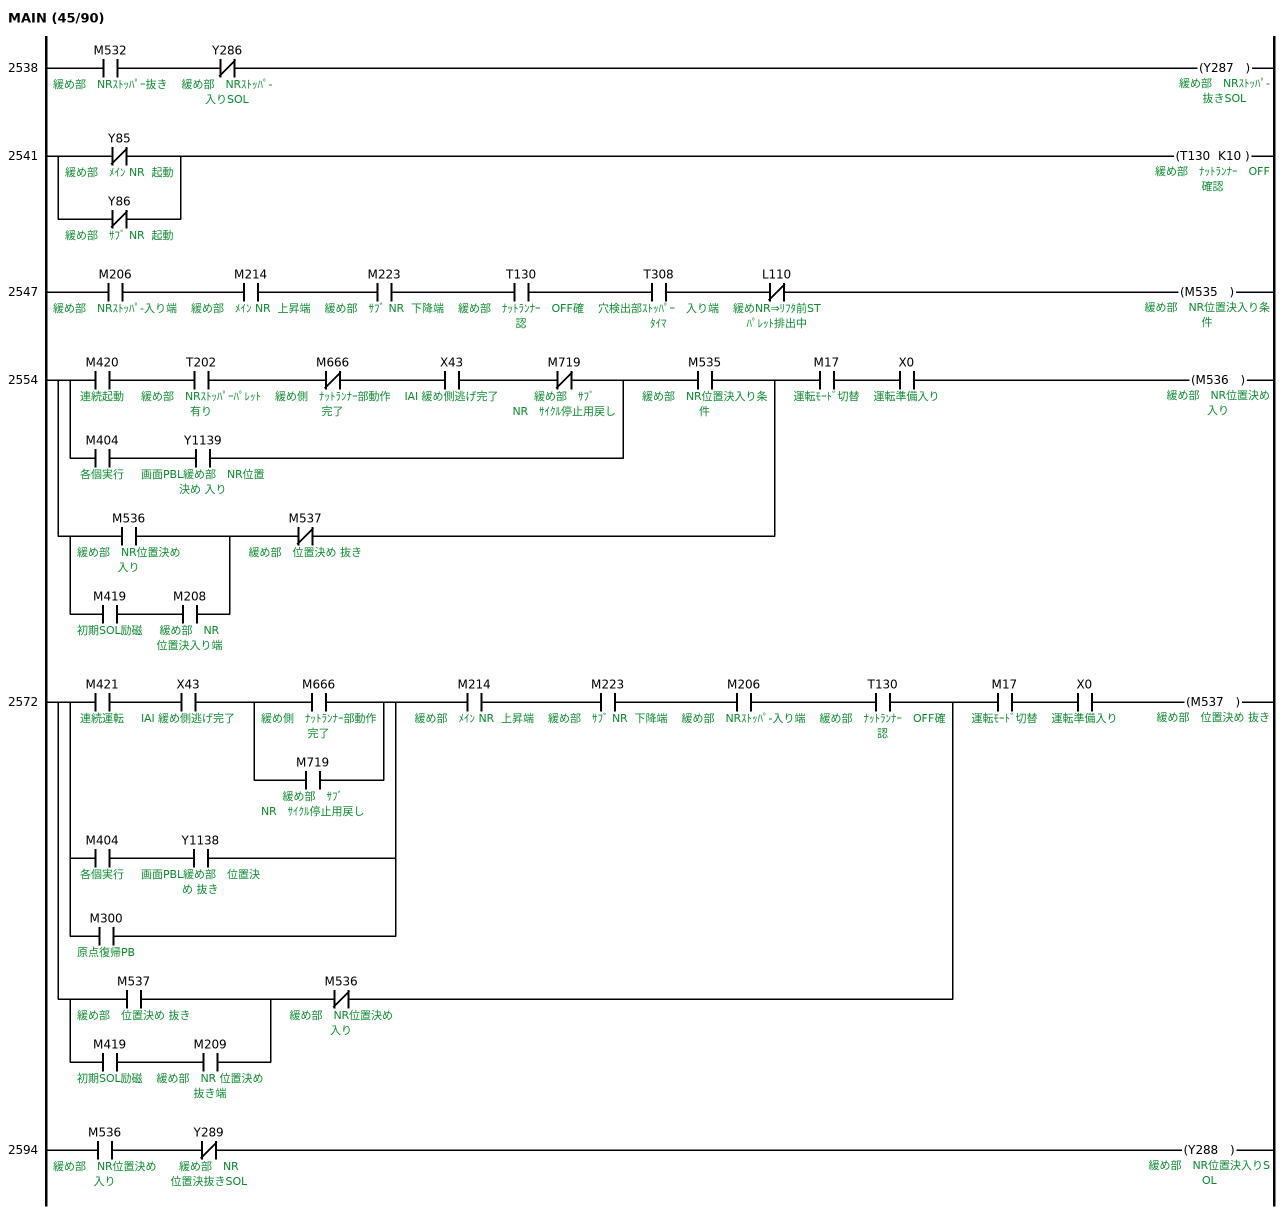
2538  LD      M532  ; 緩め部　NRｽﾄｯﾊﾟｰ抜き
      ANI     Y286  ; 緩め部　NRｽﾄｯﾊﾟ-入りSOL
      OUT     Y287  ; 緩め部　NRｽﾄｯﾊﾟ-抜きSOL
2541  LDI     Y85  ; 緩め部　ﾒｲﾝ NR  起動
      ORI     Y86  ; 緩め部　ｻﾌﾞ NR  起動
      OUT     T130 K10  ; 緩め部　ﾅｯﾄﾗﾝﾅｰ　OFF確認
2547  LD      M206  ; 緩め部　NRｽﾄｯﾊﾟ-入り端
      AND     M214  ; 緩め部　ﾒｲﾝ NR  上昇端
      AND     M223  ; 緩め部　ｻﾌﾞ NR  下降端
      AND     T130  ; 緩め部　ﾅｯﾄﾗﾝﾅｰ　OFF確認
      AND     T308  ; 穴検出部ｽﾄｯﾊﾟｰ　入り端　ﾀｲﾏ
      ANI     L110  ; 緩めNR⇒ﾘﾌﾀ前ST ﾊﾟﾚｯﾄ排出中
      OUT     M535  ; 緩め部　NR位置決入り条件
2554  LD      M420  ; 連続起動
      AND     T202  ; 緩め部　NRｽﾄｯﾊﾟｰﾊﾟﾚｯﾄ有り
      ANI     M666  ; 緩め側　ﾅｯﾄﾗﾝﾅｰ部動作完了
      AND     X43  ; IAI 緩め側逃げ完了
      ANI     M719  ; 緩め部　ｻﾌﾞ NR　ｻｲｸﾙ停止用戻し
      LD      M404  ; 各個実行
      AND     Y1139  ; 画面PBL緩め部　NR位置決め 入り
      ORB
      AND     M535  ; 緩め部　NR位置決入り条件
      LD      M536  ; 緩め部　NR位置決め 入り
      LD      M419  ; 初期SOL励磁
      AND     M208  ; 緩め部　NR 位置決入り端
      ORB
      ANI     M537  ; 緩め部　位置決め 抜き
      ORB
      AND     M17  ; 運転ﾓｰﾄﾞ切替
      AND     X0  ; 運転準備入り
      OUT     M536  ; 緩め部　NR位置決め 入り
2572  LD      M421  ; 連続運転
      AND     X43  ; IAI 緩め側逃げ完了
      LD      M666  ; 緩め側　ﾅｯﾄﾗﾝﾅｰ部動作完了
      OR      M719  ; 緩め部　ｻﾌﾞ NR　ｻｲｸﾙ停止用戻し
      ANB
      LD      M404  ; 各個実行
      AND     Y1138  ; 画面PBL緩め部　位置決め 抜き
      ORB
      OR      M300  ; 原点復帰PB
      AND     M214  ; 緩め部　ﾒｲﾝ NR  上昇端
      AND     M223  ; 緩め部　ｻﾌﾞ NR  下降端
      AND     M206  ; 緩め部　NRｽﾄｯﾊﾟ-入り端
      AND     T130  ; 緩め部　ﾅｯﾄﾗﾝﾅｰ　OFF確認
      LD      M537  ; 緩め部　位置決め 抜き
      LD      M419  ; 初期SOL励磁
      AND     M209  ; 緩め部　NR 位置決め 抜き端
      ORB
      ANI     M536  ; 緩め部　NR位置決め 入り
      ORB
      AND     M17  ; 運転ﾓｰﾄﾞ切替
      AND     X0  ; 運転準備入り
      OUT     M537  ; 緩め部　位置決め 抜き
2594  LD      M536  ; 緩め部　NR位置決め 入り
      ANI     Y289  ; 緩め部　NR 位置決抜きSOL
      OUT     Y288  ; 緩め部　NR位置決入りSOL
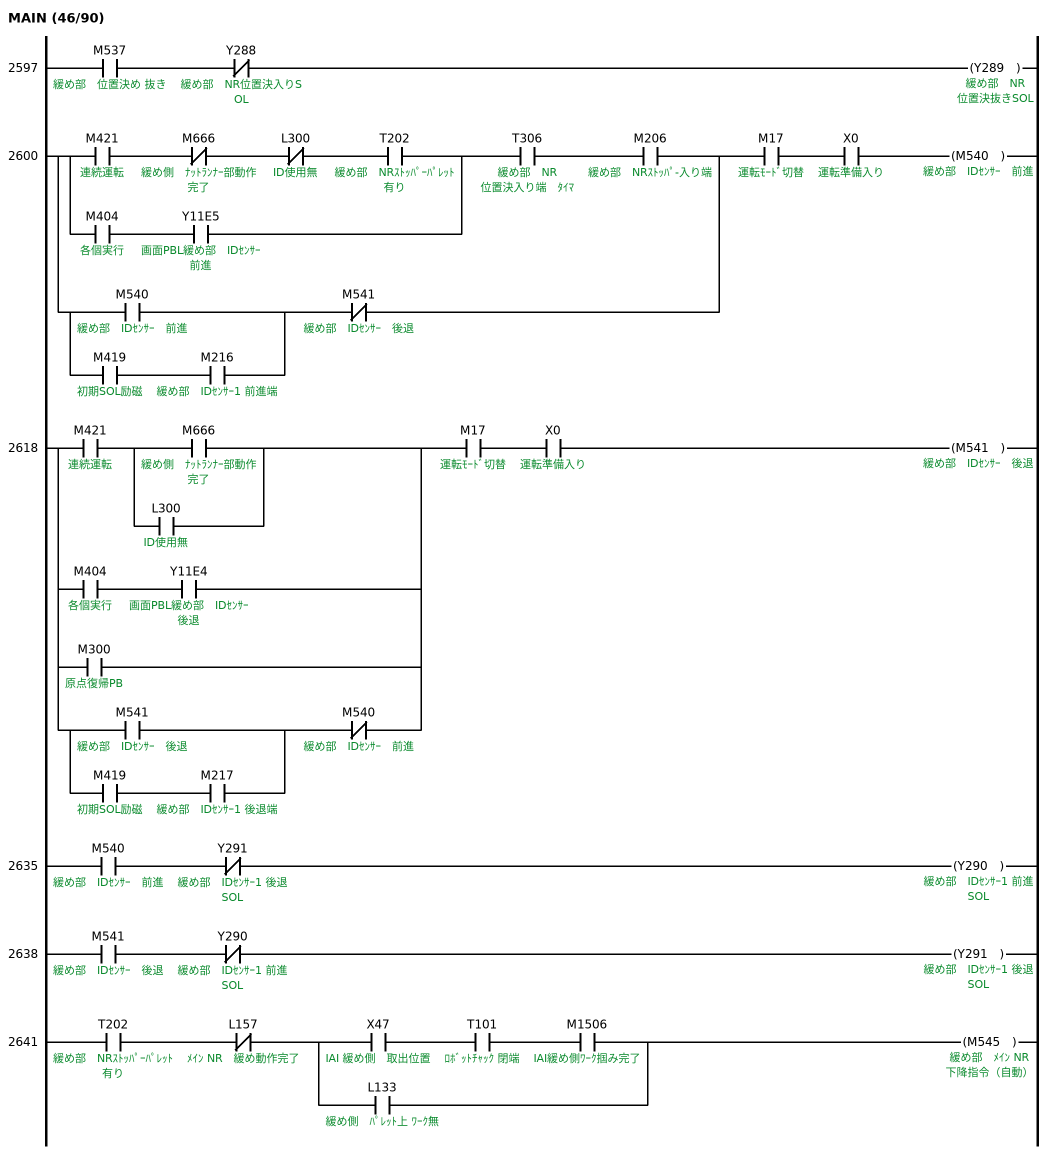
2597  LD      M537  ; 緩め部　位置決め 抜き
      ANI     Y288  ; 緩め部　NR位置決入りSOL
      OUT     Y289  ; 緩め部　NR 位置決抜きSOL
2600  LD      M421  ; 連続運転
      ANI     M666  ; 緩め側　ﾅｯﾄﾗﾝﾅｰ部動作完了
      ANI     L300  ; ID使用無
      AND     T202  ; 緩め部　NRｽﾄｯﾊﾟｰﾊﾟﾚｯﾄ有り
      LD      M404  ; 各個実行
      AND     Y11E5  ; 画面PBL緩め部　IDｾﾝｻｰ　前進
      ORB
      AND     T306  ; 緩め部　NR 位置決入り端　ﾀｲﾏ
      AND     M206  ; 緩め部　NRｽﾄｯﾊﾟ-入り端
      LD      M540  ; 緩め部　IDｾﾝｻｰ　前進
      LD      M419  ; 初期SOL励磁
      AND     M216  ; 緩め部　IDｾﾝｻｰ1 前進端
      ORB
      ANI     M541  ; 緩め部　IDｾﾝｻｰ　後退
      ORB
      AND     M17  ; 運転ﾓｰﾄﾞ切替
      AND     X0  ; 運転準備入り
      OUT     M540  ; 緩め部　IDｾﾝｻｰ　前進
2618  LD      M421  ; 連続運転
      LD      M666  ; 緩め側　ﾅｯﾄﾗﾝﾅｰ部動作完了
      OR      L300  ; ID使用無
      ANB
      LD      M404  ; 各個実行
      AND     Y11E4  ; 画面PBL緩め部　IDｾﾝｻｰ　後退
      ORB
      OR      M300  ; 原点復帰PB
      LD      M541  ; 緩め部　IDｾﾝｻｰ　後退
      LD      M419  ; 初期SOL励磁
      AND     M217  ; 緩め部　IDｾﾝｻｰ1 後退端
      ORB
      ANI     M540  ; 緩め部　IDｾﾝｻｰ　前進
      ORB
      AND     M17  ; 運転ﾓｰﾄﾞ切替
      AND     X0  ; 運転準備入り
      OUT     M541  ; 緩め部　IDｾﾝｻｰ　後退
2635  LD      M540  ; 緩め部　IDｾﾝｻｰ　前進
      ANI     Y291  ; 緩め部　IDｾﾝｻｰ1 後退 SOL
      OUT     Y290  ; 緩め部　IDｾﾝｻｰ1 前進 SOL
2638  LD      M541  ; 緩め部　IDｾﾝｻｰ　後退
      ANI     Y290  ; 緩め部　IDｾﾝｻｰ1 前進 SOL
      OUT     Y291  ; 緩め部　IDｾﾝｻｰ1 後退 SOL
2641  LD      T202  ; 緩め部　NRｽﾄｯﾊﾟｰﾊﾟﾚｯﾄ有り
      ANI     L157  ; ﾒｲﾝ NR　緩め動作完了
      LD      X47  ; IAI 緩め側　取出位置
      AND     T101  ; ﾛﾎﾞｯﾄﾁｬｯｸ 閉端
      AND     M1506  ; IAI緩め側ﾜｰｸ掴み完了
      OR      L133  ; 緩め側　ﾊﾟﾚｯﾄ上 ﾜｰｸ無
      ANB
      OUT     M545  ; 緩め部　ﾒｲﾝ NR  下降指令（自動）
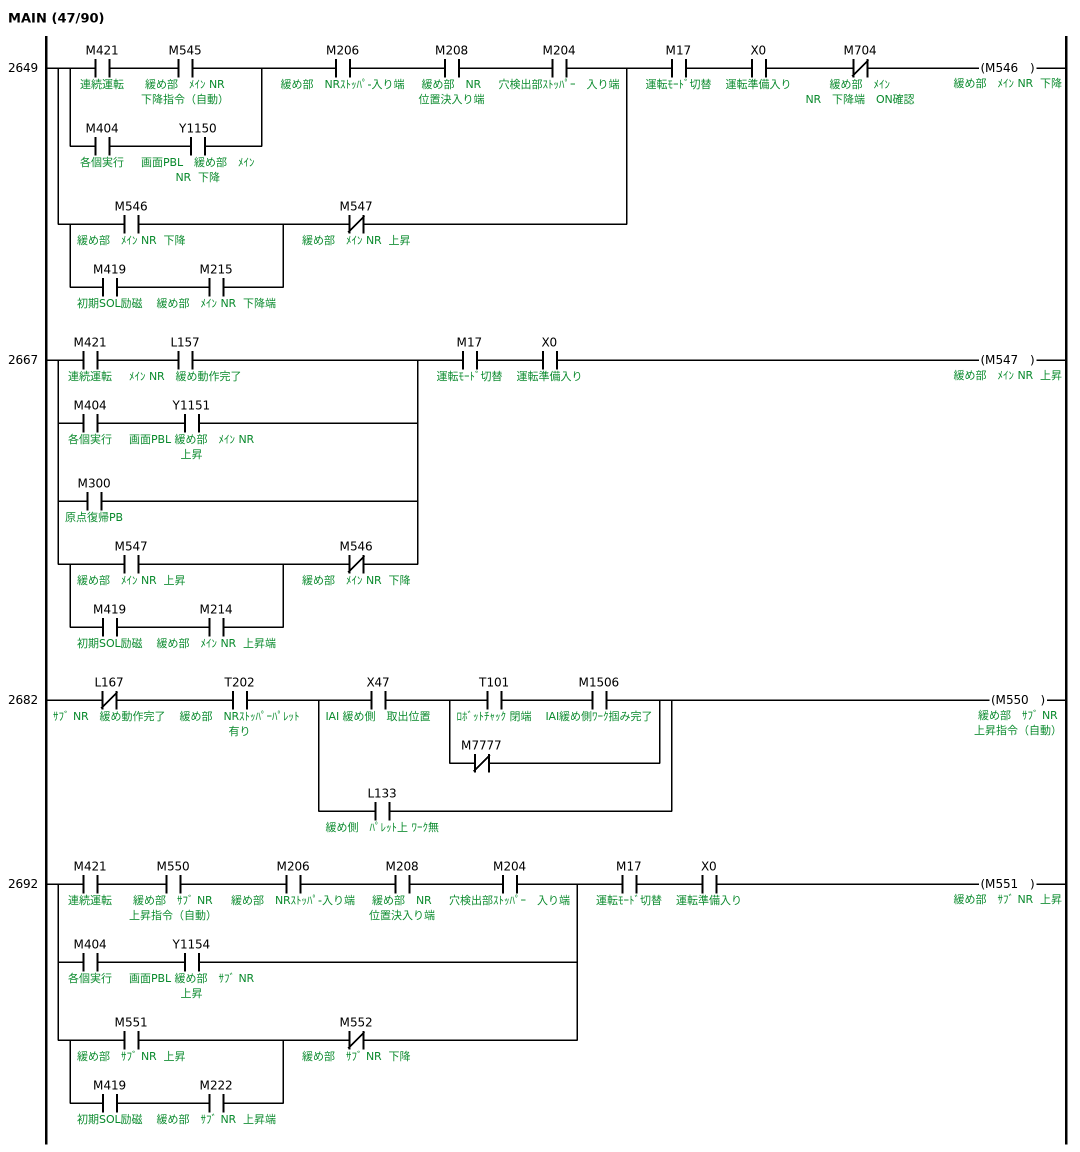
2649  LD      M421  ; 連続運転
      AND     M545  ; 緩め部　ﾒｲﾝ NR  下降指令（自動）
      LD      M404  ; 各個実行
      AND     Y1150  ; 画面PBL　緩め部　ﾒｲﾝ NR  下降
      ORB
      AND     M206  ; 緩め部　NRｽﾄｯﾊﾟ-入り端
      AND     M208  ; 緩め部　NR 位置決入り端
      AND     M204  ; 穴検出部ｽﾄｯﾊﾟｰ　入り端
      LD      M546  ; 緩め部　ﾒｲﾝ NR  下降
      LD      M419  ; 初期SOL励磁
      AND     M215  ; 緩め部　ﾒｲﾝ NR  下降端
      ORB
      ANI     M547  ; 緩め部　ﾒｲﾝ NR  上昇
      ORB
      AND     M17  ; 運転ﾓｰﾄﾞ切替
      AND     X0  ; 運転準備入り
      ANI     M704  ; 緩め部　ﾒｲﾝ NR　下降端　ON確認
      OUT     M546  ; 緩め部　ﾒｲﾝ NR  下降
2667  LD      M421  ; 連続運転
      AND     L157  ; ﾒｲﾝ NR　緩め動作完了
      LD      M404  ; 各個実行
      AND     Y1151  ; 画面PBL 緩め部　ﾒｲﾝ NR  上昇
      ORB
      OR      M300  ; 原点復帰PB
      LD      M547  ; 緩め部　ﾒｲﾝ NR  上昇
      LD      M419  ; 初期SOL励磁
      AND     M214  ; 緩め部　ﾒｲﾝ NR  上昇端
      ORB
      ANI     M546  ; 緩め部　ﾒｲﾝ NR  下降
      ORB
      AND     M17  ; 運転ﾓｰﾄﾞ切替
      AND     X0  ; 運転準備入り
      OUT     M547  ; 緩め部　ﾒｲﾝ NR  上昇
2682  LDI     L167  ; ｻﾌﾞ NR　緩め動作完了
      AND     T202  ; 緩め部　NRｽﾄｯﾊﾟｰﾊﾟﾚｯﾄ有り
      LD      X47  ; IAI 緩め側　取出位置
      LD      T101  ; ﾛﾎﾞｯﾄﾁｬｯｸ 閉端
      AND     M1506  ; IAI緩め側ﾜｰｸ掴み完了
      ORI     M7777
      ANB
      OR      L133  ; 緩め側　ﾊﾟﾚｯﾄ上 ﾜｰｸ無
      ANB
      OUT     M550  ; 緩め部　ｻﾌﾞ NR  上昇指令（自動）
2692  LD      M421  ; 連続運転
      AND     M550  ; 緩め部　ｻﾌﾞ NR  上昇指令（自動）
      AND     M206  ; 緩め部　NRｽﾄｯﾊﾟ-入り端
      AND     M208  ; 緩め部　NR 位置決入り端
      AND     M204  ; 穴検出部ｽﾄｯﾊﾟｰ　入り端
      LD      M404  ; 各個実行
      AND     Y1154  ; 画面PBL 緩め部　ｻﾌﾞ NR  上昇
      ORB
      LD      M551  ; 緩め部　ｻﾌﾞ NR  上昇
      LD      M419  ; 初期SOL励磁
      AND     M222  ; 緩め部　ｻﾌﾞ NR  上昇端
      ORB
      ANI     M552  ; 緩め部　ｻﾌﾞ NR  下降
      ORB
      AND     M17  ; 運転ﾓｰﾄﾞ切替
      AND     X0  ; 運転準備入り
      OUT     M551  ; 緩め部　ｻﾌﾞ NR  上昇
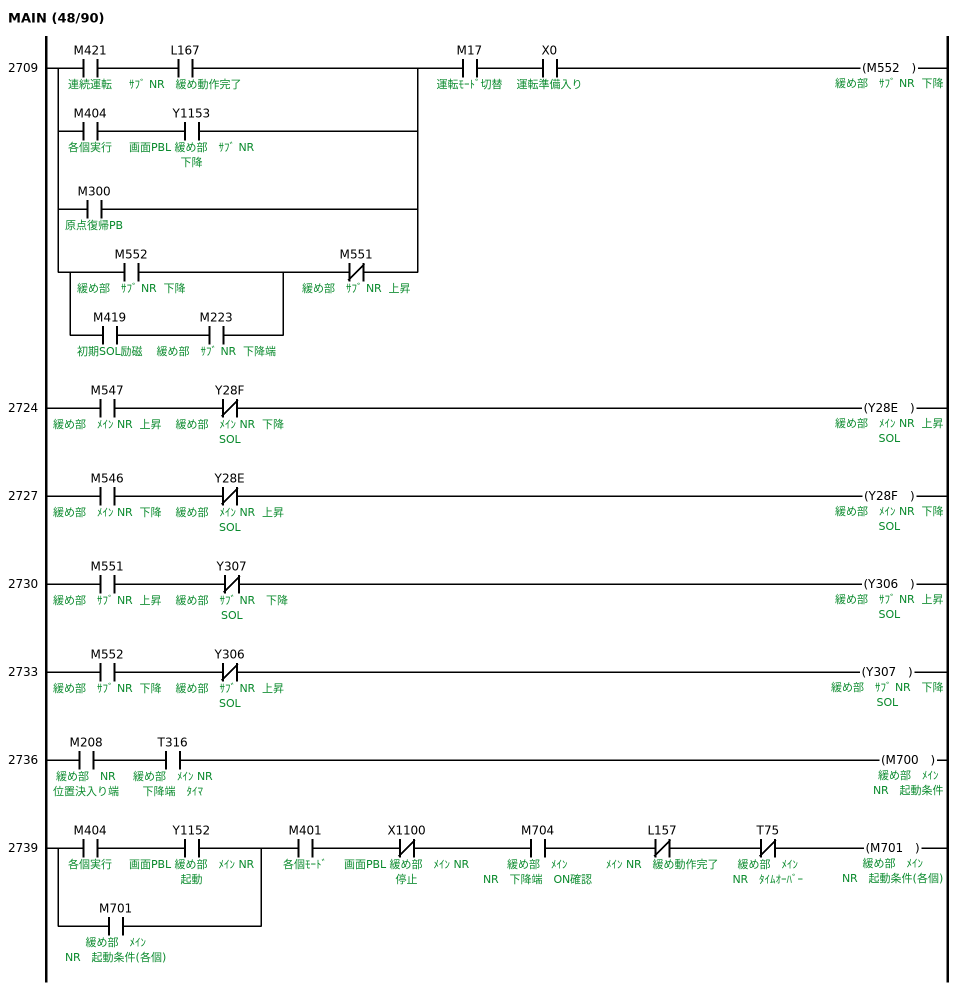
2709  LD      M421  ; 連続運転
      AND     L167  ; ｻﾌﾞ NR　緩め動作完了
      LD      M404  ; 各個実行
      AND     Y1153  ; 画面PBL 緩め部　ｻﾌﾞ NR  下降
      ORB
      OR      M300  ; 原点復帰PB
      LD      M552  ; 緩め部　ｻﾌﾞ NR  下降
      LD      M419  ; 初期SOL励磁
      AND     M223  ; 緩め部　ｻﾌﾞ NR  下降端
      ORB
      ANI     M551  ; 緩め部　ｻﾌﾞ NR  上昇
      ORB
      AND     M17  ; 運転ﾓｰﾄﾞ切替
      AND     X0  ; 運転準備入り
      OUT     M552  ; 緩め部　ｻﾌﾞ NR  下降
2724  LD      M547  ; 緩め部　ﾒｲﾝ NR  上昇
      ANI     Y28F  ; 緩め部　ﾒｲﾝ NR  下降 SOL
      OUT     Y28E  ; 緩め部　ﾒｲﾝ NR  上昇 SOL
2727  LD      M546  ; 緩め部　ﾒｲﾝ NR  下降
      ANI     Y28E  ; 緩め部　ﾒｲﾝ NR  上昇 SOL
      OUT     Y28F  ; 緩め部　ﾒｲﾝ NR  下降 SOL
2730  LD      M551  ; 緩め部　ｻﾌﾞ NR  上昇
      ANI     Y307  ; 緩め部　ｻﾌﾞ NR　下降 SOL
      OUT     Y306  ; 緩め部　ｻﾌﾞ NR  上昇 SOL
2733  LD      M552  ; 緩め部　ｻﾌﾞ NR  下降
      ANI     Y306  ; 緩め部　ｻﾌﾞ NR  上昇 SOL
      OUT     Y307  ; 緩め部　ｻﾌﾞ NR　下降 SOL
2736  LD      M208  ; 緩め部　NR 位置決入り端
      AND     T316  ; 緩め部　ﾒｲﾝ NR  下降端　ﾀｲﾏ
      OUT     M700  ; 緩め部　ﾒｲﾝ NR　起動条件
2739  LD      M404  ; 各個実行
      AND     Y1152  ; 画面PBL 緩め部　ﾒｲﾝ NR  起動
      OR      M701  ; 緩め部　ﾒｲﾝ NR　起動条件(各個)
      AND     M401  ; 各個ﾓｰﾄﾞ
      ANI     X1100  ; 画面PBL 緩め部　ﾒｲﾝ NR  停止
      AND     M704  ; 緩め部　ﾒｲﾝ NR　下降端　ON確認
      ANI     L157  ; ﾒｲﾝ NR　緩め動作完了
      ANI     T75  ; 緩め部　ﾒｲﾝ NR　ﾀｲﾑｵｰﾊﾞｰ
      OUT     M701  ; 緩め部　ﾒｲﾝ NR　起動条件(各個)
